KUKA KRL program: MyProgram_022().src

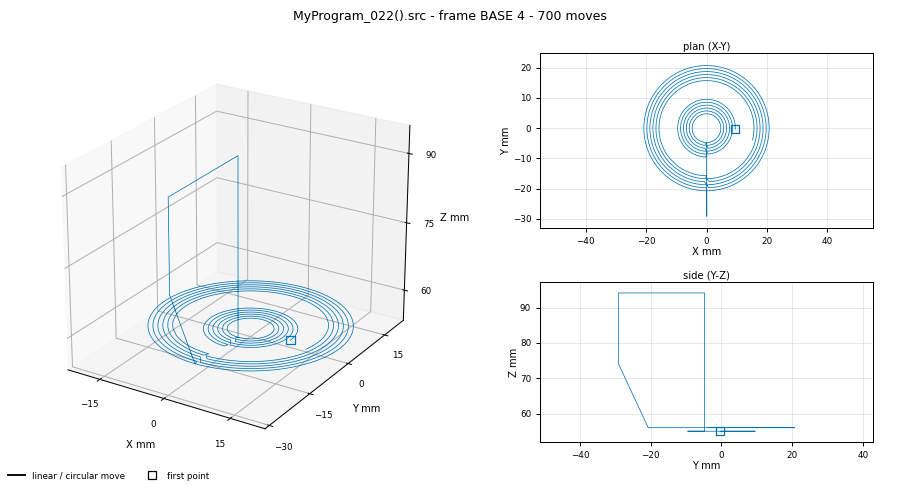
[picture p0: tool path of MyProgram_022().src in frame BASE 4, 700 of 700 moves have a stored position in this frame; points joined in program order, loops and branches not executed]
&ACCESS RVP
&REL 1
&PARAM TEMPLATE = C:\KRC\Roboter\Template\vorgabe
&PARAM EDITMASK = *
DEF MyProgram_022()
; ---- Setting reference (Base) ----
$BASE = BASE_DATA[4]

; --------------------------
; ---- Setting tool (TCP) ----
$TOOL = TOOL_DATA[3]
; --------------------------

$VEL.CP = VEL_APROX_PRINT
Startdeposition()
$VEL.CP = VEL_PRINT
LIN {X 9.5437,Y -0.3407,Z 55,A -8.3961,B 24.5035,C -3.2675,E1 24.8669,E2 -269.4642} C_DIS
LIN {X 9.52,Y 0.7548,Z 55,A -1.6453,B 24.5009,C -3.2888,E1 24.8659,E2 -276.2255} C_DIS
LIN {X 9.3724,Y 1.8321,Z 55,A 5.8885,B 24.4976,C -3.3147,E1 24.8622,E2 -283.7766} C_DIS
LIN {X 8.9196,Y 3.4119,Z 55,A 15.084,B 24.4945,C -3.3389,E1 24.8541,E2 -292.9776} C_DIS
LIN {X 8.1843,Y 4.9212,Z 55,A 24.5802,B 24.4915,C -3.3621,E1 24.8417,E2 -302.4789} C_DIS
LIN {X 7.5338,Y 5.8685,Z 55,A 31.3136,B 24.4895,C -3.3777,E1 24.8306,E2 -309.2166} C_DIS
LIN {X 6.8523,Y 6.6485,Z 55,A 37.0507,B 24.4881,C -3.3886,E1 24.8199,E2 -314.9542} C_DIS
LIN {X 6.0078,Y 7.4234,Z 55,A 44.3227,B 24.4861,C -3.4035,E1 24.8046,E2 -322.233} C_DIS
LIN {X 5.0818,Y 8.0855,Z 55,A 51.1975,B 24.4847,C -3.4144,E1 24.7887,E2 -329.1106} C_DIS
LIN {X 4.1712,Y 8.5908,Z 55,A 57.4744,B 24.4837,C -3.4223,E1 24.7731,E2 -335.3889} C_DIS
LIN {X 3.3474,Y 8.9438,Z 55,A 62.8052,B 24.483,C -3.4273,E1 24.7593,E2 -340.7196} C_DIS
LIN {X 2.409,Y 9.2406,Z 55,A 69.1697,B 24.4823,C -3.4329,E1 24.7422,E2 -347.0869} C_DIS
LIN {X 1.1691,Y 9.477,Z 55,A 76.1197,B 24.4823,C -3.4331,E1 24.723,E2 -354.0304} C_DIS
LIN {X 0.1545,Y 9.5485,Z 55,A 82.3576,B 24.4823,C -3.4331,E1 24.7056,E2 -360.2665} C_DIS
LIN {X -1.2836,Y 9.4632,Z 55,A 91.4292,B 24.4826,C -3.4303,E1 24.6804,E2 -369.3357} C_DIS
LIN {X -2.5093,Y 9.2143,Z 55,A 98.8876,B 24.4835,C -3.4234,E1 24.6602,E2 -376.7878} C_DIS
LIN {X -3.3779,Y 8.9324,Z 55,A 105.3226,B 24.4842,C -3.4184,E1 24.6434,E2 -383.2239} C_DIS
LIN {X -4.9252,Y 8.1819,Z 55,A 114.2089,B 24.4867,C -3.3995,E1 24.6215,E2 -392.0897} C_DIS
LIN {X -5.8293,Y 7.5644,Z 55,A 121.6467,B 24.4882,C -3.3875,E1 24.6048,E2 -399.525} C_DIS
LIN {X -6.7767,Y 6.7285,Z 55,A 128.6516,B 24.4905,C -3.3699,E1 24.5905,E2 -406.5164} C_DIS
LIN {X -7.5818,Y 5.8012,Z 55,A 134.4735,B 24.493,C -3.3508,E1 24.5801,E2 -412.319} C_DIS
LIN {X -8.0674,Y 5.1105,Z 55,A 141.4999,B 24.4946,C -3.338,E1 24.5691,E2 -419.3498} C_DIS
LIN {X -8.6788,Y 3.9781,Z 55,A 147.4247,B 24.4974,C -3.3158,E1 24.5615,E2 -425.2526} C_DIS
LIN {X -9.0093,Y 3.1669,Z 55,A 154.8449,B 24.4994,C -3.3005,E1 24.5541,E2 -432.6779} C_DIS
LIN {X -9.3639,Y 1.875,Z 55,A 161.7964,B 24.5025,C -3.2759,E1 24.5495,E2 -439.6111} C_DIS
LIN {X -9.529,Y 0.6276,Z 55,A 171.0146,B 24.5054,C -3.2526,E1 24.5469,E2 -448.8287} C_DIS
LIN {X -9.5121,Y -0.8487,Z 55,A 178.9892,B 24.5088,C -3.2253,E1 24.548,E2 -456.7858} C_DIS
LIN {X -9.3498,Y -1.944,Z 55,A -174.6947,B 24.5112,C -3.2053,E1 24.551,E2 -463.0913} C_DIS
LIN {X -9.078,Y -2.965,Z 55,A -167.6269,B 24.5135,C -3.187,E1 24.5566,E2 -470.1561} C_DIS
LIN {X -8.6807,Y -3.9802,Z 55,A -161.2388,B 24.5157,C -3.169,E1 24.5636,E2 -476.5362} C_DIS
LIN {X -8.1263,Y -5.0163,Z 55,A -154.1121,B 24.5179,C -3.1509,E1 24.5735,E2 -483.6566} C_DIS
LIN {X -7.4885,Y -5.9263,Z 55,A -147.3718,B 24.5198,C -3.1353,E1 24.5848,E2 -490.392} C_DIS
LIN {X -6.6668,Y -6.8377,Z 55,A -139.7416,B 24.5215,C -3.1203,E1 24.5996,E2 -498.0193} C_DIS
LIN {X -5.7118,Y -7.6497,Z 55,A -133.1323,B 24.5233,C -3.1057,E1 24.6139,E2 -504.6186} C_DIS
LIN {X -4.7809,Y -8.267,Z 55,A -125.9127,B 24.5243,C -3.0968,E1 24.631,E2 -511.8397} C_DIS
LIN {X -3.8134,Y -8.7552,Z 55,A -118.9983,B 24.5251,C -3.0904,E1 24.6485,E2 -518.7563} C_DIS
LIN {X -2.6205,Y -9.1833,Z 55,A -111.5476,B 24.5258,C -3.0845,E1 24.6683,E2 -526.2062} C_DIS
LIN {X -1.4624,Y -9.4371,Z 55,A -104.4401,B 24.5261,C -3.082,E1 24.6878,E2 -533.3153} C_DIS
LIN {X -0.2812,Y -9.5456,Z 55,A -97.8601,B 24.5263,C -3.0804,E1 24.7061,E2 -539.8939} C_DIS
LIN {X -0.2812,Y -9.5456,Z 55,A -97.8601,B 24.5263,C -3.0804,E1 24.7061,E2 -539.8939} C_DIS
Enddeposition()
LIN {X 0.0484,Y -8.5882,Z 55,A -96.4156,B 19.666,C -2.0295,E1 19.7657,E2 -540.06} C_DIS
Startdeposition()
$VEL.CP = VEL_PRINT
LIN {X -1.0617,Y -8.5255,Z 55,A -105.0334,B 19.6663,C -2.0274,E1 19.7417,E2 -531.431} C_DIS
LIN {X -2.1331,Y -8.3222,Z 55,A -111.7699,B 19.6658,C -2.0316,E1 19.7233,E2 -524.6964} C_DIS
LIN {X -2.9014,Y -8.0865,Z 55,A -117.4774,B 19.6655,C -2.0353,E1 19.7082,E2 -518.986} C_DIS
LIN {X -3.626,Y -7.7883,Z 55,A -122.789,B 19.6649,C -2.0407,E1 19.6947,E2 -513.6739} C_DIS
LIN {X -4.5351,Y -7.2969,Z 55,A -130.0587,B 19.664,C -2.0498,E1 19.6772,E2 -506.4028} C_DIS
LIN {X -5.617,Y -6.5006,Z 55,A -138.2989,B 19.6625,C -2.0653,E1 19.6591,E2 -498.1697} C_DIS
LIN {X -6.3065,Y -5.8281,Z 55,A -144.638,B 19.6612,C -2.0782,E1 19.6467,E2 -491.8342} C_DIS
LIN {X -6.8045,Y -5.2401,Z 55,A -149.8115,B 19.66,C -2.0896,E1 19.6376,E2 -486.6633} C_DIS
LIN {X -7.4508,Y -4.2776,Z 55,A -158.3349,B 19.658,C -2.1086,E1 19.6249,E2 -478.1405} C_DIS
LIN {X -7.8893,Y -3.4012,Z 55,A -165.4977,B 19.6562,C -2.1262,E1 19.6167,E2 -470.9797} C_DIS
LIN {X -8.3397,Y -2.0642,Z 55,A -174.2614,B 19.6535,C -2.1523,E1 19.6097,E2 -462.2282} C_DIS
LIN {X -8.5403,Y -0.9049,Z 55,A 179.7232,B 19.6512,C -2.1738,E1 19.6071,E2 -456.2308} C_DIS
LIN {X -8.5918,Y -0.0576,Z 55,A 171.3138,B 19.6492,C -2.1929,E1 19.6063,E2 -447.813} C_DIS
LIN {X -8.5069,Y 1.2012,Z 55,A 164.3732,B 19.6466,C -2.2167,E1 19.6081,E2 -440.8896} C_DIS
LIN {X -8.3384,Y 2.0688,Z 55,A 156.7921,B 19.6446,C -2.2355,E1 19.6128,E2 -433.307} C_DIS
LIN {X -7.8607,Y 3.4667,Z 55,A 148.6266,B 19.6416,C -2.2623,E1 19.6208,E2 -425.162} C_DIS
LIN {X -7.4985,Y 4.1927,Z 55,A 141.6224,B 19.6399,C -2.2779,E1 19.63,E2 -418.1563} C_DIS
LIN {X -6.649,Y 5.4408,Z 55,A 133.1113,B 19.6371,C -2.3025,E1 19.6439,E2 -409.665} C_DIS
LIN {X -6.1281,Y 6.021,Z 55,A 125.7768,B 19.6358,C -2.3146,E1 19.6581,E2 -402.3256} C_DIS
LIN {X -4.7675,Y 7.1472,Z 55,A 114.9917,B 19.6332,C -2.3374,E1 19.6819,E2 -391.5581} C_DIS
LIN {X -4.0838,Y 7.5577,Z 55,A 109.5222,B 19.6322,C -2.3457,E1 19.6953,E2 -386.0929} C_DIS
LIN {X -2.9018,Y 8.0863,Z 55,A 100.8347,B 19.631,C -2.3565,E1 19.7177,E2 -377.4126} C_DIS
LIN {X -1.6334,Y 8.434,Z 55,A 92.4272,B 19.6301,C -2.3643,E1 19.7405,E2 -369.0136} C_DIS
LIN {X -0.6223,Y 8.5687,Z 55,A 85.3058,B 19.6298,C -2.3669,E1 19.7602,E2 -361.8945} C_DIS
LIN {X 0.509,Y 8.5714,Z 55,A 78.3367,B 19.6296,C -2.3687,E1 19.7797,E2 -354.9324} C_DIS
LIN {X 1.2791,Y 8.4924,Z 55,A 73.1686,B 19.6297,C -2.3675,E1 19.794,E2 -349.7659} C_DIS
LIN {X 2.0387,Y 8.3424,Z 55,A 68.0068,B 19.63,C -2.3649,E1 19.808,E2 -344.6055} C_DIS
LIN {X 3.1694,Y 7.9849,Z 55,A 60.3912,B 19.6307,C -2.3592,E1 19.8281,E2 -336.9923} C_DIS
LIN {X 4.1301,Y 7.5333,Z 55,A 51.4713,B 19.6324,C -2.3444,E1 19.8503,E2 -328.0604} C_DIS
LIN {X 5.3942,Y 6.6869,Z 55,A 44.1822,B 19.633,C -2.3388,E1 19.8669,E2 -320.7874} C_DIS
LIN {X 6.1554,Y 5.9934,Z 55,A 35.7616,B 19.6352,C -2.3192,E1 19.8841,E2 -312.3536} C_DIS
LIN {X 6.7864,Y 5.2679,Z 55,A 28.6991,B 19.6372,C -2.3022,E1 19.8965,E2 -305.2831} C_DIS
LIN {X 7.5014,Y 4.1881,Z 55,A 21.2861,B 19.6389,C -2.2866,E1 19.9074,E2 -297.8727} C_DIS
LIN {X 7.8951,Y 3.3879,Z 55,A 15.4697,B 19.6406,C -2.2715,E1 19.9143,E2 -292.0525} C_DIS
LIN {X 8.2732,Y 2.3161,Z 55,A 7.2455,B 19.6433,C -2.2472,E1 19.9215,E2 -283.8168} C_DIS
LIN {X 8.491,Y 1.2828,Z 55,A 0.8671,B 19.6452,C -2.2301,E1 19.9248,E2 -277.4363} C_DIS
LIN {X 8.5896,Y 0.1713,Z 55,A -7.1351,B 19.6479,C -2.2051,E1 19.9261,E2 -269.4218} C_DIS
LIN {X 8.5419,Y -0.9196,Z 55,A -14.0427,B 19.65,C -2.1853,E1 19.9248,E2 -262.5087} C_DIS
LIN {X 8.3771,Y -1.906,Z 55,A -21.1303,B 19.6523,C -2.1634,E1 19.9209,E2 -255.4101} C_DIS
LIN {X 8.0567,Y -2.9832,Z 55,A -28.7401,B 19.6547,C -2.1411,E1 19.9142,E2 -247.7903} C_DIS
LIN {X 7.587,Y -4.0309,Z 55,A -35.9207,B 19.6566,C -2.1223,E1 19.9054,E2 -240.6039} C_DIS
LIN {X 6.9736,Y -5.0179,Z 55,A -45.1996,B 19.6594,C -2.0953,E1 19.8908,E2 -231.3045} C_DIS
LIN {X 5.6333,Y -6.4865,Z 55,A -56.5929,B 19.6616,C -2.0736,E1 19.8684,E2 -219.91} C_DIS
LIN {X 4.5247,Y -7.3028,Z 55,A -67.0354,B 19.6638,C -2.0518,E1 19.8443,E2 -209.4489} C_DIS
LIN {X 3.1306,Y -8.0001,Z 55,A -77.5224,B 19.6653,C -2.0372,E1 19.8175,E2 -198.952} C_DIS
LIN {X 1.7735,Y -8.4063,Z 55,A -86.5252,B 19.666,C -2.03,E1 19.7932,E2 -189.9452} C_DIS
LIN {X 0.493,Y -8.5769,Z 55,A -94.5546,B 19.6662,C -2.0275,E1 19.7709,E2 -181.9148} C_DIS
LIN {X 0.493,Y -8.5769,Z 55,A -94.5546,B 19.6662,C -2.0275,E1 19.7709,E2 -181.9148} C_DIS
Enddeposition()
LIN {X -0.0072,Y -7.6328,Z 55,A -91.0932,B 14.7927,C -1.2124,E1 14.8521,E2 -184.2665} C_DIS
Startdeposition()
$VEL.CP = VEL_PRINT
LIN {X 1.7414,Y -7.4315,Z 55,A -79.0266,B 14.7923,C -1.2183,E1 14.8852,E2 -196.3334} C_DIS
LIN {X 3.0947,Y -6.9771,Z 55,A -69.7981,B 14.7916,C -1.2267,E1 14.9093,E2 -205.56} C_DIS
LIN {X 3.8118,Y -6.6129,Z 55,A -64.1101,B 14.7909,C -1.2346,E1 14.9234,E2 -211.2506} C_DIS
LIN {X 4.7649,Y -5.9629,Z 55,A -52.7906,B 14.7889,C -1.2595,E1 14.9488,E2 -222.596} C_DIS
LIN {X 5.9068,Y -4.8341,Z 55,A -40.8403,B 14.7866,C -1.2863,E1 14.9711,E2 -234.5569} C_DIS
LIN {X 6.931,Y -3.1967,Z 55,A -28.3133,B 14.7841,C -1.3158,E1 14.9882,E2 -247.0842} C_DIS
LIN {X 7.2359,Y -2.4292,Z 55,A -21.4776,B 14.7823,C -1.3357,E1 14.9947,E2 -253.9303} C_DIS
LIN {X 7.5213,Y -1.3,Z 55,A -13.0631,B 14.7802,C -1.3594,E1 14.9996,E2 -262.3507} C_DIS
LIN {X 7.6295,Y -0.2251,Z 55,A -5.4007,B 14.7783,C -1.381,E1 15.001,E2 -270.0173} C_DIS
LIN {X 7.5606,Y 1.0475,Z 55,A 4.7584,B 14.7755,C -1.4111,E1 14.9984,E2 -280.188} C_DIS
LIN {X 7.3346,Y 2.1124,Z 55,A 12.6105,B 14.7735,C -1.4325,E1 14.993,E2 -288.0437} C_DIS
LIN {X 6.904,Y 3.2548,Z 55,A 21.287,B 14.7714,C -1.4546,E1 14.9837,E2 -296.7226} C_DIS
LIN {X 6.4679,Y 4.053,Z 55,A 28.2666,B 14.7697,C -1.4719,E1 14.9738,E2 -303.7065} C_DIS
LIN {X 5.86,Y 4.8857,Z 55,A 35.0672,B 14.7683,C -1.4858,E1 14.9623,E2 -310.5044} C_DIS
LIN {X 5.403,Y 5.3885,Z 55,A 40.3436,B 14.7672,C -1.4968,E1 14.9521,E2 -315.7833} C_DIS
LIN {X 4.5877,Y 6.1003,Z 55,A 48.6669,B 14.7657,C -1.5118,E1 14.9342,E2 -324.1091} C_DIS
LIN {X 3.6389,Y 6.7096,Z 55,A 58.0991,B 14.7643,C -1.5264,E1 14.9116,E2 -333.5471} C_DIS
LIN {X 2.5598,Y 7.1908,Z 55,A 66.5015,B 14.7635,C -1.534,E1 14.8898,E2 -341.9457} C_DIS
LIN {X 1.3106,Y 7.5193,Z 55,A 76.1296,B 14.763,C -1.5391,E1 14.8636,E2 -351.5707} C_DIS
LIN {X 0.2159,Y 7.6256,Z 55,A 83.5677,B 14.763,C -1.5388,E1 14.8429,E2 -359.0012} C_DIS
LIN {X -0.8816,Y 7.5817,Z 55,A 91.5987,B 14.7633,C -1.5362,E1 14.8206,E2 -367.0266} C_DIS
LIN {X -1.6402,Y 7.4545,Z 55,A 98.3351,B 14.7636,C -1.5333,E1 14.8021,E2 -373.7643} C_DIS
LIN {X -2.5722,Y 7.1863,Z 55,A 105.734,B 14.7643,C -1.5262,E1 14.7825,E2 -381.1586} C_DIS
LIN {X -3.6086,Y 6.7255,Z 55,A 113.7963,B 14.7654,C -1.5147,E1 14.7623,E2 -389.2118} C_DIS
LIN {X -4.467,Y 6.1826,Z 55,A 121.4415,B 14.7667,C -1.5019,E1 14.7445,E2 -396.8508} C_DIS
LIN {X -5.1004,Y 5.6736,Z 55,A 127.6071,B 14.7679,C -1.49,E1 14.7314,E2 -403.0111} C_DIS
LIN {X -5.6752,Y 5.0991,Z 55,A 133.8696,B 14.7692,C -1.4766,E1 14.7194,E2 -409.2685} C_DIS
LIN {X -6.305,Y 4.302,Z 55,A 141.9263,B 14.771,C -1.4579,E1 14.7061,E2 -417.3199} C_DIS
LIN {X -6.8966,Y 3.2703,Z 55,A 151.3038,B 14.7733,C -1.434,E1 14.6939,E2 -426.6908} C_DIS
LIN {X -7.3324,Y 2.1063,Z 55,A 159.9509,B 14.7757,C -1.409,E1 14.6862,E2 -435.3257} C_DIS
LIN {X -7.5725,Y 0.9578,Z 55,A 168.9473,B 14.7781,C -1.3833,E1 14.6818,E2 -444.3148} C_DIS
LIN {X -7.6314,Y 0.1435,Z 55,A 175.5205,B 14.7797,C -1.3649,E1 14.681,E2 -450.8849} C_DIS
LIN {X -7.5817,Y -0.8637,Z 55,A -177.4519,B 14.7816,C -1.3438,E1 14.6825,E2 -457.9037} C_DIS
LIN {X -7.4779,Y -1.5155,Z 55,A -172.4272,B 14.7829,C -1.3297,E1 14.685,E2 -462.9251} C_DIS
LIN {X -7.3187,Y -2.1561,Z 55,A -167.5507,B 14.7841,C -1.3161,E1 14.6886,E2 -467.7976} C_DIS
LIN {X -7.1055,Y -2.7807,Z 55,A -162.5731,B 14.7852,C -1.3027,E1 14.6933,E2 -472.7722} C_DIS
LIN {X -6.6528,Y -3.7418,Z 55,A -153.6372,B 14.787,C -1.2816,E1 14.7047,E2 -481.7088} C_DIS
LIN {X -6.2826,Y -4.3348,Z 55,A -147.702,B 14.7881,C -1.2688,E1 14.714,E2 -487.6455} C_DIS
LIN {X -5.4108,Y -5.3837,Z 55,A -138.4398,B 14.7898,C -1.2482,E1 14.7312,E2 -496.899} C_DIS
LIN {X -4.5966,Y -6.0937,Z 55,A -129.9493,B 14.791,C -1.2341,E1 14.7496,E2 -505.3903} C_DIS
LIN {X -3.8307,Y -6.602,Z 55,A -122.8606,B 14.7918,C -1.2244,E1 14.7664,E2 -512.4797} C_DIS
LIN {X -2.8961,Y -7.0619,Z 55,A -115.5853,B 14.7924,C -1.2159,E1 14.7849,E2 -519.7524} C_DIS
LIN {X -2.0683,Y -7.3434,Z 55,A -109.3433,B 14.7929,C -1.2108,E1 14.8015,E2 -525.9939} C_DIS
LIN {X -1.0315,Y -7.5626,Z 55,A -99.7498,B 14.7929,C -1.2099,E1 14.8279,E2 -535.6} C_DIS
LIN {X -0.0072,Y -7.6328,Z 55,A -95.8758,B 14.7934,C -1.2042,E1 14.8386,E2 -539.4534} C_DIS
Enddeposition()
LIN {X -0.0072,Y -7.6328,Z 55,A -95.8758,B 14.7934,C -1.2042,E1 14.8386,E2 -539.4534} C_DIS
Startdeposition()
$VEL.CP = VEL_PRINT
LIN {X -0.5513,Y -6.6453,Z 55,A -99.3031,B 9.8862,C -0.5743,E1 9.8872,E2 -534.9699} C_DIS
LIN {X -1.4265,Y -6.52,Z 55,A -108.8863,B 9.8861,C -0.5765,E1 9.8609,E2 -525.3735} C_DIS
LIN {X -2.7177,Y -6.0958,Z 55,A -119.3612,B 9.8855,C -0.5868,E1 9.8336,E2 -514.9021} C_DIS
LIN {X -3.4112,Y -5.7368,Z 55,A -126.4444,B 9.885,C -0.5957,E1 9.8164,E2 -507.8162} C_DIS
LIN {X -4.2862,Y -5.1161,Z 55,A -135.5205,B 9.884,C -0.6107,E1 9.7963,E2 -498.7408} C_DIS
LIN {X -5.0009,Y -4.4131,Z 55,A -143.9478,B 9.883,C -0.6275,E1 9.78,E2 -490.3155} C_DIS
LIN {X -5.6735,Y -3.5155,Z 55,A -154.2169,B 9.8815,C -0.6504,E1 9.7637,E2 -480.0455} C_DIS
LIN {X -6.1829,Y -2.5134,Z 55,A -164.5095,B 9.8798,C -0.6761,E1 9.7518,E2 -469.7535} C_DIS
LIN {X -6.5159,Y -1.4238,Z 55,A -173.0169,B 9.8782,C -0.7003,E1 9.7455,E2 -461.2563} C_DIS
LIN {X -6.629,Y -0.7484,Z 55,A -179.2232,B 9.8769,C -0.7174,E1 9.7431,E2 -455.0517} C_DIS
LIN {X -6.6704,Y -0.0648,Z 55,A 174.6774,B 9.8757,C -0.7346,E1 9.7425,E2 -448.9549} C_DIS
LIN {X -6.6273,Y 0.7901,Z 55,A 166.5401,B 9.874,C -0.757,E1 9.7445,E2 -440.8189} C_DIS
LIN {X -6.3943,Y 1.901,Z 55,A 156.9959,B 9.872,C -0.7837,E1 9.7508,E2 -431.2824} C_DIS
LIN {X -6.1141,Y 2.6653,Z 55,A 150.0872,B 9.8705,C -0.8022,E1 9.758,E2 -424.3791} C_DIS
LIN {X -5.7439,Y 3.3901,Z 55,A 142.9913,B 9.869,C -0.82,E1 9.7675,E2 -417.288} C_DIS
LIN {X -5.2892,Y 4.0652,Z 55,A 135.855,B 9.8677,C -0.8365,E1 9.7791,E2 -410.1563} C_DIS
LIN {X -4.7541,Y 4.6787,Z 55,A 128.7619,B 9.8664,C -0.8515,E1 9.7925,E2 -403.0681} C_DIS
LIN {X -3.8851,Y 5.427,Z 55,A 117.8688,B 9.8648,C -0.8702,E1 9.8164,E2 -392.178} C_DIS
LIN {X -2.9088,Y 6.0071,Z 55,A 108.4824,B 9.8636,C -0.8834,E1 9.8394,E2 -382.7998} C_DIS
LIN {X -1.9263,Y 6.3903,Z 55,A 99.5045,B 9.8628,C -0.8922,E1 9.863,E2 -373.828} C_DIS
LIN {X -0.8857,Y 6.6117,Z 55,A 92.459,B 9.8623,C -0.898,E1 9.8823,E2 -366.7966} C_DIS
LIN {X 0.1331,Y 6.6728,Z 55,A 80.869,B 9.8623,C -0.8972,E1 9.9146,E2 -355.1986} C_DIS
LIN {X 1.2683,Y 6.5482,Z 55,A 72.5953,B 9.8625,C -0.8955,E1 9.9374,E2 -346.9354} C_DIS
LIN {X 1.9117,Y 6.3913,Z 55,A 66.8902,B 9.8629,C -0.8915,E1 9.9528,E2 -341.2319} C_DIS
LIN {X 3.0336,Y 5.945,Z 55,A 55.2257,B 9.8641,C -0.8775,E1 9.9826,E2 -329.5632} C_DIS
LIN {X 3.8966,Y 5.4188,Z 55,A 46.0037,B 9.8654,C -0.8626,E1 10.0038,E2 -320.3392} C_DIS
LIN {X 4.9697,Y 4.4553,Z 55,A 34.8499,B 9.8672,C -0.8418,E1 10.026,E2 -309.1902} C_DIS
LIN {X 5.472,Y 3.8144,Z 55,A 28.6234,B 9.8683,C -0.8284,E1 10.0363,E2 -302.9662} C_DIS
LIN {X 5.818,Y 3.2625,Z 55,A 23.1367,B 9.8694,C -0.8152,E1 10.0442,E2 -297.4784} C_DIS
LIN {X 6.1096,Y 2.68,Z 55,A 17.5975,B 9.8706,C -0.8012,E1 10.0507,E2 -291.9376} C_DIS
LIN {X 6.3418,Y 2.0713,Z 55,A 12.2288,B 9.8717,C -0.7871,E1 10.0557,E2 -286.5677} C_DIS
LIN {X 6.582,Y 1.1054,Z 55,A 3.0945,B 9.8737,C -0.7613,E1 10.0611,E2 -277.4261} C_DIS
LIN {X 6.6738,Y 0.0305,Z 55,A -7.2201,B 9.8759,C -0.7312,E1 10.0623,E2 -267.1005} C_DIS
LIN {X 6.5795,Y -1.1203,Z 55,A -18.0928,B 9.8782,C -0.6997,E1 10.0578,E2 -256.2161} C_DIS
LIN {X 6.045,Y -2.829,Z 55,A -31.9199,B 9.8807,C -0.6638,E1 10.044,E2 -242.3863} C_DIS
LIN {X 5.2656,Y -4.1012,Z 55,A -43.2424,B 9.8824,C -0.6376,E1 10.0264,E2 -231.0624} C_DIS
LIN {X 4.795,Y -4.6426,Z 55,A -51.3115,B 9.8835,C -0.6188,E1 10.0109,E2 -222.9781} C_DIS
LIN {X 3.4915,Y -5.6883,Z 55,A -63.9968,B 9.8848,C -0.5978,E1 9.9822,E2 -210.2916} C_DIS
LIN {X 2.6709,Y -6.1105,Z 55,A -71.3878,B 9.8854,C -0.5883,E1 9.9637,E2 -202.8983} C_DIS
LIN {X 1.9793,Y -6.3683,Z 55,A -77.5808,B 9.8858,C -0.582,E1 9.9473,E2 -196.7021} C_DIS
LIN {X 1.2637,Y -6.5499,Z 55,A -84.0144,B 9.886,C -0.5772,E1 9.9298,E2 -190.2642} C_DIS
LIN {X 0.5322,Y -6.6495,Z 55,A -90.4765,B 9.8862,C -0.5743,E1 9.9118,E2 -183.7981} C_DIS
LIN {X 0.5322,Y -6.6495,Z 55,A -90.4765,B 9.8862,C -0.5743,E1 9.9118,E2 -183.7981} C_DIS
Enddeposition()
LIN {X -0.0091,Y -5.7118,Z 55,A -2.8836,B 0,C 0,E1 0.1598,E2 -269.9283} C_DIS
Startdeposition()
$VEL.CP = VEL_PRINT
LIN {X 0.9619,Y -5.6271,Z 55,A -2.8445,B 0,C 0,E1 0.1598,E2 -269.9283} C_DIS
LIN {X 1.7206,Y -5.4461,Z 55,A -2.8089,B 0,C 0,E1 0.1598,E2 -269.9282} C_DIS
LIN {X 2.4463,Y -5.1598,Z 55,A -2.77,B 0,C 0,E1 0.1598,E2 -269.9282} C_DIS
LIN {X 3.127,Y -4.7788,Z 55,A -2.7288,B 0,C 0,E1 0.1598,E2 -269.9282} C_DIS
LIN {X 4.0215,Y -4.0615,Z 55,A -2.6651,B 0,C 0,E1 0.1598,E2 -269.9282} C_DIS
LIN {X 4.6904,Y -3.2657,Z 55,A -2.6064,B 0,C 0,E1 0.1598,E2 -269.9282} C_DIS
LIN {X 5.1397,Y -2.4895,Z 55,A -2.5568,B 0,C 0,E1 0.1598,E2 -269.9282} C_DIS
LIN {X 5.4534,Y -1.6925,Z 55,A -2.5112,B 0,C 0,E1 0.1598,E2 -269.9282} C_DIS
LIN {X 5.6446,Y -0.8577,Z 55,A -2.4685,B 0,C 0,E1 0.1598,E2 -269.9282} C_DIS
LIN {X 5.7096,Y -0.0038,Z 55,A -2.4296,B 0,C 0,E1 0.1598,E2 -269.9281} C_DIS
LIN {X 5.6161,Y 1.0625,Z 55,A -2.3872,B 0,C 0,E1 0.1598,E2 -269.9284} C_DIS
LIN {X 5.3029,Y 2.1179,Z 55,A -2.3537,B 0,C 0,E1 0.1598,E2 -269.9283} C_DIS
LIN {X 4.959,Y 2.8274,Z 55,A -2.3364,B 0,C 0,E1 0.1598,E2 -269.9279} C_DIS
LIN {X 4.5235,Y 3.4846,Z 55,A -2.3245,B 0,C 0,E1 0.1598,E2 -269.9278} C_DIS
LIN {X 4.0015,Y 4.0757,Z 55,A -2.3186,B 0,C 0,E1 0.1598,E2 -269.9278} C_DIS
LIN {X 3.4014,Y 4.5875,Z 55,A -2.3189,B 0,C 0,E1 0.1598,E2 -269.9277} C_DIS
LIN {X 2.7366,Y 5.0113,Z 55,A -2.3254,B 0,C 0,E1 0.1598,E2 -269.9277} C_DIS
LIN {X 1.7186,Y 5.4511,Z 55,A -2.3442,B 0,C 0,E1 0.1598,E2 -269.9277} C_DIS
LIN {X 0.5579,Y 5.6885,Z 55,A -2.377,B 0,C 0,E1 0.1598,E2 -269.9277} C_DIS
LIN {X -0.385,Y 5.6987,Z 55,A -2.4114,B 0,C 0,E1 0.1598,E2 -269.9277} C_DIS
LIN {X -1.1326,Y 5.5975,Z 55,A -2.4432,B 0,C 0,E1 0.1598,E2 -269.9277} C_DIS
LIN {X -1.8604,Y 5.4,Z 55,A -2.4785,B 0,C 0,E1 0.1598,E2 -269.9277} C_DIS
LIN {X -2.5543,Y 5.1047,Z 55,A -2.5166,B 0,C 0,E1 0.1598,E2 -269.9278} C_DIS
LIN {X -3.2057,Y 4.7249,Z 55,A -2.5567,B 0,C 0,E1 0.1598,E2 -269.9279} C_DIS
LIN {X -3.8016,Y 4.2624,Z 55,A -2.5982,B 0,C 0,E1 0.1598,E2 -269.928} C_DIS
LIN {X -4.3298,Y 3.7239,Z 55,A -2.6405,B 0,C 0,E1 0.1598,E2 -269.928} C_DIS
LIN {X -4.7804,Y 3.1193,Z 55,A -2.6827,B 0,C 0,E1 0.1598,E2 -269.9282} C_DIS
LIN {X -5.1513,Y 2.4628,Z 55,A -2.7242,B 0,C 0,E1 0.1598,E2 -269.9282} C_DIS
LIN {X -5.431,Y 1.7624,Z 55,A -2.7641,B 0,C 0,E1 0.1598,E2 -269.9284} C_DIS
LIN {X -5.6177,Y 1.0317,Z 55,A -2.802,B 0,C 0,E1 0.1598,E2 -269.9284} C_DIS
LIN {X -5.7035,Y 0.2823,Z 55,A -2.8369,B 0,C 0,E1 0.1598,E2 -269.9285} C_DIS
LIN {X -5.69,Y -0.4718,Z 55,A -2.8684,B 0,C 0,E1 0.1598,E2 -269.9285} C_DIS
LIN {X -5.541,Y -1.4026,Z 55,A -2.9022,B 0,C 0,E1 0.1598,E2 -269.9288} C_DIS
LIN {X -4.946,Y -2.8649,Z 55,A -2.9418,B 0,C 0,E1 0.1598,E2 -269.9295} C_DIS
LIN {X -4.4029,Y -3.645,Z 55,A -2.9555,B 0,C 0,E1 0.1598,E2 -269.9291} C_DIS
LIN {X -3.4666,Y -4.5443,Z 55,A -2.9596,B 0,C 0,E1 0.1598,E2 -269.9288} C_DIS
LIN {X -2.4461,Y -5.1659,Z 55,A -2.9488,B 0,C 0,E1 0.1598,E2 -269.9286} C_DIS
LIN {X -1.3162,Y -5.5622,Z 55,A -2.9243,B 0,C 0,E1 0.1598,E2 -269.9284} C_DIS
LIN {X -0.5027,Y -5.6894,Z 55,A -2.9,B 0,C 0,E1 0.1598,E2 -269.9284} C_DIS
LIN {X -0.5027,Y -5.6894,Z 55,A -2.9,B 0,C 0,E1 0.1598,E2 -269.9283} C_DIS
Enddeposition()
LIN {X -0.0164,Y -4.7573,Z 55,A -2.841,B 0,C 0,E1 0.1598,E2 -269.9295} C_DIS
Startdeposition()
$VEL.CP = VEL_PRINT
LIN {X -0.8506,Y -4.6765,Z 55,A -2.8694,B 0,C 0,E1 0.1598,E2 -269.9283} C_DIS
LIN {X -1.5,Y -4.5096,Z 55,A -2.8862,B 0,C 0,E1 0.1598,E2 -269.9283} C_DIS
LIN {X -2.1197,Y -4.2534,Z 55,A -2.898,B 0,C 0,E1 0.1598,E2 -269.9283} C_DIS
LIN {X -2.6968,Y -3.9121,Z 55,A -2.9046,B 0,C 0,E1 0.1598,E2 -269.9283} C_DIS
LIN {X -3.2199,Y -3.4929,Z 55,A -2.906,B 0,C 0,E1 0.1598,E2 -269.9284} C_DIS
LIN {X -3.6802,Y -3.0058,Z 55,A -2.9021,B 0,C 0,E1 0.1598,E2 -269.9284} C_DIS
LIN {X -4.0666,Y -2.458,Z 55,A -2.893,B 0,C 0,E1 0.1598,E2 -269.9284} C_DIS
LIN {X -4.372,Y -1.8613,Z 55,A -2.8788,B 0,C 0,E1 0.1598,E2 -269.9284} C_DIS
LIN {X -4.5913,Y -1.2278,Z 55,A -2.86,B 0,C 0,E1 0.1598,E2 -269.9284} C_DIS
LIN {X -4.7168,Y -0.5691,Z 55,A -2.8366,B 0,C 0,E1 0.1598,E2 -269.9284} C_DIS
LIN {X -4.7518,Y 0.1003,Z 55,A -2.8094,B 0,C 0,E1 0.1598,E2 -269.9284} C_DIS
LIN {X -4.6905,Y 0.768,Z 55,A -2.7788,B 0,C 0,E1 0.1598,E2 -269.9284} C_DIS
LIN {X -4.5362,Y 1.4205,Z 55,A -2.7455,B 0,C 0,E1 0.1598,E2 -269.9284} C_DIS
LIN {X -4.2904,Y 2.0444,Z 55,A -2.71,B 0,C 0,E1 0.1598,E2 -269.9282} C_DIS
LIN {X -3.9574,Y 2.6262,Z 55,A -2.673,B 0,C 0,E1 0.1598,E2 -269.9282} C_DIS
LIN {X -3.5516,Y 3.1598,Z 55,A -2.6355,B 0,C 0,E1 0.1598,E2 -269.9281} C_DIS
LIN {X -3.0711,Y 3.6275,Z 55,A -2.5979,B 0,C 0,E1 0.1598,E2 -269.9281} C_DIS
LIN {X -2.5298,Y 4.0232,Z 55,A -2.5612,B 0,C 0,E1 0.1598,E2 -269.9279} C_DIS
LIN {X -1.9382,Y 4.3386,Z 55,A -2.526,B 0,C 0,E1 0.1598,E2 -269.9279} C_DIS
LIN {X -1.3083,Y 4.568,Z 55,A -2.4931,B 0,C 0,E1 0.1598,E2 -269.9278} C_DIS
LIN {X -0.6525,Y 4.7067,Z 55,A -2.4631,B 0,C 0,E1 0.1598,E2 -269.9278} C_DIS
LIN {X 0.0164,Y 4.7515,Z 55,A -2.4365,B 0,C 0,E1 0.1598,E2 -269.9277} C_DIS
LIN {X 0.6849,Y 4.7021,Z 55,A -2.414,B 0,C 0,E1 0.1598,E2 -269.9277} C_DIS
LIN {X 1.3398,Y 4.5588,Z 55,A -2.3959,B 0,C 0,E1 0.1598,E2 -269.9277} C_DIS
LIN {X 1.9677,Y 4.3241,Z 55,A -2.3827,B 0,C 0,E1 0.1598,E2 -269.9277} C_DIS
LIN {X 2.5574,Y 4.0054,Z 55,A -2.3745,B 0,C 0,E1 0.1598,E2 -269.9277} C_DIS
LIN {X 3.096,Y 3.6061,Z 55,A -2.3717,B 0,C 0,E1 0.1598,E2 -269.9277} C_DIS
LIN {X 3.5733,Y 3.1352,Z 55,A -2.3741,B 0,C 0,E1 0.1598,E2 -269.9277} C_DIS
LIN {X 3.9773,Y 2.5999,Z 55,A -2.382,B 0,C 0,E1 0.1598,E2 -269.9277} C_DIS
LIN {X 4.3039,Y 2.0145,Z 55,A -2.3949,B 0,C 0,E1 0.1598,E2 -269.9278} C_DIS
LIN {X 4.546,Y 1.3893,Z 55,A -2.4127,B 0,C 0,E1 0.1598,E2 -269.9278} C_DIS
LIN {X 4.6955,Y 0.7357,Z 55,A -2.435,B 0,C 0,E1 0.1598,E2 -269.9279} C_DIS
LIN {X 4.7525,Y 0.0675,Z 55,A -2.4615,B 0,C 0,E1 0.1598,E2 -269.9279} C_DIS
LIN {X 4.7136,Y -0.6018,Z 55,A -2.4915,B 0,C 0,E1 0.1598,E2 -269.928} C_DIS
LIN {X 4.5819,Y -1.2591,Z 55,A -2.5244,B 0,C 0,E1 0.1598,E2 -269.928} C_DIS
LIN {X 4.359,Y -1.8913,Z 55,A -2.5596,B 0,C 0,E1 0.1598,E2 -269.928} C_DIS
LIN {X 4.0496,Y -2.486,Z 55,A -2.5964,B 0,C 0,E1 0.1598,E2 -269.928} C_DIS
LIN {X 3.6587,Y -3.0304,Z 55,A -2.634,B 0,C 0,E1 0.1598,E2 -269.928} C_DIS
LIN {X 3.1965,Y -3.516,Z 55,A -2.6717,B 0,C 0,E1 0.1598,E2 -269.9281} C_DIS
LIN {X 2.6698,Y -3.9308,Z 55,A -2.7088,B 0,C 0,E1 0.1598,E2 -269.9281} C_DIS
LIN {X 2.0903,Y -4.268,Z 55,A -2.7445,B 0,C 0,E1 0.1598,E2 -269.9281} C_DIS
LIN {X 1.469,Y -4.5201,Z 55,A -2.7781,B 0,C 0,E1 0.1598,E2 -269.9281} C_DIS
LIN {X 0.8184,Y -4.6823,Z 55,A -2.8089,B 0,C 0,E1 0.1598,E2 -269.9281} C_DIS
LIN {X -0.0164,Y -4.7573,Z 55,A -2.8427,B 0,C 0,E1 0.1598,E2 -269.9282} C_DIS
Enddeposition()
LIN {X -0.0164,Y -4.7573,Z 60,A -2.8323,B 0,C 0,E1 0.1598,E2 -269.928} C_DIS
LIN {X -0.0164,Y -4.7571,Z 75,A -2.8055,B 0,C 0,E1 0.1598,E2 -269.927} C_DIS
LIN {X -0.0164,Y -4.7571,Z 94.1262,A -2.7793,B 0,C 0,E1 0.1598,E2 -269.9267} C_DIS
LIN {X 0.0643,Y -29.1728,Z 94.1262,A -97.2324,B 24.8219,C -3.0777,E1 25.0005,E2 -180.429} C_DIS
LIN {X 0.0643,Y -29.1728,Z 74.1262,A -96.9044,B 24.8376,C -2.94,E1 25.0005,E2 -180.429} C_DIS
LIN {X 0.0569,Y -22.8335,Z 60.5315,A -96.9447,B 24.8357,C -2.9569,E1 25.0005,E2 -180.429} C_DIS
LIN {X 0.0545,Y -20.7204,Z 56,A -96.9596,B 24.835,C -2.9632,E1 25.0005,E2 -180.429} C_DIS
Startdeposition()
$VEL.CP = VEL_PRINT
LIN {X 1.2873,Y -20.6848,Z 56,A -92.294,B 24.8338,C -2.9734,E1 25.0136,E2 -185.1177} C_DIS
LIN {X 3.0514,Y -20.4994,Z 56,A -87.4914,B 24.8336,C -2.9757,E1 25.0269,E2 -189.9219} C_DIS
LIN {X 4.6788,Y -20.1899,Z 56,A -82.799,B 24.833,C -2.9805,E1 25.0397,E2 -194.6198} C_DIS
LIN {X 6.3703,Y -19.7216,Z 56,A -77.9231,B 24.8324,C -2.9861,E1 25.0528,E2 -199.5004} C_DIS
LIN {X 7.9462,Y -19.1409,Z 56,A -73.5263,B 24.8319,C -2.9903,E1 25.0642,E2 -203.8974} C_DIS
LIN {X 9.4639,Y -18.4379,Z 56,A -68.7364,B 24.831,C -2.999,E1 25.0762,E2 -208.6953} C_DIS
LIN {X 11.0059,Y -17.5611,Z 56,A -63.8256,B 24.83,C -3.0078,E1 25.088,E2 -213.6119} C_DIS
LIN {X 12.456,Y -16.5641,Z 56,A -58.9873,B 24.8289,C -3.0173,E1 25.099,E2 -218.4557} C_DIS
LIN {X 13.8006,Y -15.4617,Z 56,A -54.1932,B 24.8277,C -3.0278,E1 25.1092,E2 -223.2559} C_DIS
LIN {X 15.0293,Y -14.2706,Z 56,A -49.5505,B 24.8265,C -3.0382,E1 25.1183,E2 -227.9035} C_DIS
LIN {X 16.1542,Y -12.9835,Z 56,A -44.8179,B 24.8251,C -3.0502,E1 25.1268,E2 -232.6429} C_DIS
LIN {X 17.2,Y -11.5623,Z 56,A -39.9191,B 24.8236,C -3.0634,E1 25.1347,E2 -237.5491} C_DIS
LIN {X 18.0989,Y -10.0971,Z 56,A -35.2338,B 24.8221,C -3.0761,E1 25.1413,E2 -242.2403} C_DIS
LIN {X 18.8655,Y -8.5803,Z 56,A -30.7037,B 24.8207,C -3.088,E1 25.1467,E2 -246.7744} C_DIS
LIN {X 19.4528,Y -7.1494,Z 56,A -26.3854,B 24.8192,C -3.1012,E1 25.1511,E2 -251.0999} C_DIS
LIN {X 19.9411,Y -5.6456,Z 56,A -21.9648,B 24.8176,C -3.115,E1 25.1547,E2 -255.528} C_DIS
LIN {X 20.3331,Y -4.0119,Z 56,A -17.4801,B 24.8161,C -3.1277,E1 25.1573,E2 -260.0168} C_DIS
LIN {X 20.5717,Y -2.5177,Z 56,A -13.1742,B 24.8144,C -3.142,E1 25.159,E2 -264.3311} C_DIS
LIN {X 20.7114,Y -0.7464,Z 56,A -8.943,B 24.8134,C -3.1505,E1 25.1597,E2 -268.5573} C_DIS
LIN {X 20.7189,Y 0.5147,Z 56,A -4.8529,B 24.8113,C -3.1674,E1 25.1597,E2 -272.6631} C_DIS
LIN {X 20.5986,Y 2.2843,Z 56,A -0.1749,B 24.8098,C -3.1802,E1 25.1585,E2 -277.3438} C_DIS
LIN {X 20.3685,Y 3.8281,Z 56,A 4.2815,B 24.8081,C -3.1947,E1 25.1564,E2 -281.8084} C_DIS
LIN {X 19.974,Y 5.5276,Z 56,A 9.0641,B 24.8064,C -3.2086,E1 25.1531,E2 -286.5964} C_DIS
LIN {X 19.4261,Y 7.2209,Z 56,A 13.8036,B 24.8049,C -3.221,E1 25.1487,E2 -291.3385} C_DIS
LIN {X 18.8401,Y 8.6363,Z 56,A 18.0556,B 24.8034,C -3.2328,E1 25.144,E2 -295.5954} C_DIS
LIN {X 18.0989,Y 10.0971,Z 56,A 22.6686,B 24.8019,C -3.2457,E1 25.1379,E2 -300.2145} C_DIS
LIN {X 17.1824,Y 11.5883,Z 56,A 27.501,B 24.8004,C -3.2577,E1 25.1306,E2 -305.0513} C_DIS
LIN {X 16.1542,Y 12.9835,Z 56,A 32.2543,B 24.799,C -3.2686,E1 25.1225,E2 -309.8078} C_DIS
LIN {X 15.0101,Y 14.2908,Z 56,A 37.0404,B 24.7978,C -3.2788,E1 25.1135,E2 -314.5971} C_DIS
LIN {X 13.7299,Y 15.5248,Z 56,A 41.9265,B 24.7966,C -3.2882,E1 25.1034,E2 -319.4855} C_DIS
LIN {X 12.4057,Y 16.6019,Z 56,A 46.6548,B 24.7956,C -3.2965,E1 25.093,E2 -324.2163} C_DIS
LIN {X 10.9794,Y 17.5777,Z 56,A 51.3848,B 24.7947,C -3.3034,E1 25.082,E2 -328.9472} C_DIS
LIN {X 9.4639,Y 18.4379,Z 56,A 56.2186,B 24.7939,C -3.3099,E1 25.0701,E2 -333.7824} C_DIS
LIN {X 7.8676,Y 19.1736,Z 56,A 60.8958,B 24.7934,C -3.3136,E1 25.0581,E2 -338.4571} C_DIS
LIN {X 6.3703,Y 19.7216,Z 56,A 65.453,B 24.7928,C -3.3184,E1 25.0461,E2 -343.0167} C_DIS
LIN {X 4.6788,Y 20.1899,Z 56,A 70.2628,B 24.7925,C -3.3208,E1 25.0331,E2 -347.8252} C_DIS
LIN {X 2.9949,Y 20.5075,Z 56,A 74.9908,B 24.7923,C -3.3223,E1 25.02,E2 -352.5517} C_DIS
LIN {X 1.2709,Y 20.6858,Z 56,A 79.7919,B 24.7923,C -3.3227,E1 25.0067,E2 -357.3512} C_DIS
LIN {X -0.46,Y 20.72,Z 56,A 84.5553,B 24.7924,C -3.3216,E1 24.9934,E2 -362.1118} C_DIS
LIN {X -2.1548,Y 20.6126,Z 56,A 89.3204,B 24.7926,C -3.3199,E1 24.9801,E2 -366.8752} C_DIS
LIN {X -3.8967,Y 20.3553,Z 56,A 94.192,B 24.7931,C -3.3164,E1 24.9667,E2 -371.7433} C_DIS
LIN {X -5.6456,Y 19.9411,Z 56,A 99.0777,B 24.7937,C -3.3112,E1 24.9536,E2 -376.6235} C_DIS
LIN {X -7.2363,Y 19.4203,Z 56,A 103.79,B 24.7944,C -3.306,E1 24.9412,E2 -381.3328} C_DIS
LIN {X -8.8612,Y 18.7353,Z 56,A 108.5563,B 24.7953,C -3.2984,E1 24.929,E2 -386.0924} C_DIS
LIN {X -10.239,Y 18.0193,Z 56,A 113.0452,B 24.7961,C -3.2923,E1 24.918,E2 -390.5794} C_DIS
LIN {X -11.7563,Y 17.0681,Z 56,A 117.9752,B 24.7973,C -3.283,E1 24.9065,E2 -395.5032} C_DIS
LIN {X -13.1479,Y 16.0207,Z 56,A 122.808,B 24.7985,C -3.2731,E1 24.8959,E2 -400.3302} C_DIS
LIN {X -14.464,Y 14.8434,Z 56,A 127.6385,B 24.7999,C -3.2618,E1 24.8861,E2 -405.1533} C_DIS
LIN {X -15.5924,Y 13.6528,Z 56,A 132.2799,B 24.8012,C -3.2513,E1 24.8774,E2 -409.7901} C_DIS
LIN {X -16.6815,Y 12.2985,Z 56,A 137.1615,B 24.8027,C -3.2392,E1 24.8691,E2 -414.666} C_DIS
LIN {X -17.6478,Y 10.8671,Z 56,A 141.9796,B 24.8042,C -3.2264,E1 24.8618,E2 -419.4777} C_DIS
LIN {X -18.512,Y 9.3182,Z 56,A 146.7863,B 24.806,C -3.2121,E1 24.8555,E2 -424.2757} C_DIS
LIN {X -19.1736,Y 7.8676,Z 56,A 151.1687,B 24.8075,C -3.1991,E1 24.8507,E2 -428.6511} C_DIS
LIN {X -19.7216,Y 6.3703,Z 56,A 155.7672,B 24.809,C -3.1866,E1 24.8465,E2 -433.2458} C_DIS
LIN {X -20.1899,Y 4.6788,Z 56,A 160.6442,B 24.8108,C -3.1718,E1 24.8432,E2 -438.116} C_DIS
LIN {X -20.5075,Y 2.9949,Z 56,A 165.3845,B 24.8126,C -3.1571,E1 24.841,E2 -442.8492} C_DIS
LIN {X -20.6858,Y 1.2709,Z 56,A 170.2217,B 24.8143,C -3.1424,E1 24.8399,E2 -447.6801} C_DIS
LIN {X -20.7189,Y -0.5147,Z 56,A 175.2425,B 24.8161,C -3.1273,E1 24.8399,E2 -452.6952} C_DIS
LIN {X -20.5986,Y -2.2843,Z 56,A 179.9885,B 24.818,C -3.1117,E1 24.8411,E2 -457.4321} C_DIS
LIN {X -20.3685,Y -3.8281,Z 56,A -175.4913,B 24.8194,C -3.0994,E1 24.8432,E2 -461.9497} C_DIS
LIN {X -19.974,Y -5.5276,Z 56,A -170.6418,B 24.8211,C -3.0852,E1 24.8466,E2 -466.7935} C_DIS
LIN {X -19.4261,Y -7.2209,Z 56,A -165.8138,B 24.8227,C -3.0707,E1 24.851,E2 -471.6143} C_DIS
LIN {X -18.8358,Y -8.6455,Z 56,A -161.3496,B 24.824,C -3.0598,E1 24.856,E2 -476.0769} C_DIS
LIN {X -18.0193,Y -10.239,Z 56,A -156.3699,B 24.8255,C -3.0469,E1 24.8626,E2 -481.052} C_DIS
LIN {X -17.0681,Y -11.7563,Z 56,A -151.4328,B 24.8269,C -3.0346,E1 24.8701,E2 -485.9844} C_DIS
LIN {X -16.0103,Y -13.1606,Z 56,A -146.5699,B 24.8282,C -3.0233,E1 24.8785,E2 -490.8434} C_DIS
LIN {X -14.8434,Y -14.464,Z 56,A -141.7685,B 24.8294,C -3.0129,E1 24.8877,E2 -495.6409} C_DIS
LIN {X -13.6528,Y -15.5924,Z 56,A -137.1326,B 24.8303,C -3.0047,E1 24.8972,E2 -500.2757} C_DIS
LIN {X -12.2985,Y -16.6815,Z 56,A -132.2609,B 24.8312,C -2.9967,E1 24.908,E2 -505.1462} C_DIS
LIN {X -10.8582,Y -17.6531,Z 56,A -127.4456,B 24.832,C -2.9896,E1 24.9193,E2 -509.96} C_DIS
LIN {X -9.3182,Y -18.512,Z 56,A -122.6677,B 24.8328,C -2.9829,E1 24.9311,E2 -514.7352} C_DIS
LIN {X -7.8676,Y -19.1736,Z 56,A -118.3049,B 24.8333,C -2.9781,E1 24.9423,E2 -519.0968} C_DIS
LIN {X -6.3703,Y -19.7216,Z 56,A -113.7304,B 24.8336,C -2.9756,E1 24.9544,E2 -523.6742} C_DIS
LIN {X -4.6788,Y -20.1899,Z 56,A -108.8821,B 24.8339,C -2.973,E1 24.9675,E2 -528.523} C_DIS
LIN {X -2.9944,Y -20.5076,Z 56,A -104.1726,B 24.8341,C -2.9714,E1 24.9805,E2 -533.2333} C_DIS
LIN {X -1.2709,Y -20.6858,Z 56,A -99.3709,B 24.8341,C -2.9714,E1 24.9938,E2 -538.0369} C_DIS
LIN {X 0.0545,Y -20.7204,Z 56,A -96.9596,B 24.835,C -2.9631,E1 25.0005,E2 -540.4289} C_DIS
Enddeposition()
LIN {X 0.0545,Y -20.7204,Z 56,A -96.9596,B 24.835,C -2.9631,E1 25.0005,E2 -540.4289} C_DIS
Startdeposition()
$VEL.CP = VEL_PRINT
LIN {X -0.0881,Y -19.7268,Z 56,A -98.5569,B 24.834,C -2.9724,E1 24.9961,E2 -538.8536} C_DIS
LIN {X -1.8243,Y -19.6424,Z 56,A -103.6074,B 24.834,C -2.9724,E1 24.982,E2 -533.8011} C_DIS
LIN {X -3.5089,Y -19.4123,Z 56,A -108.5479,B 24.8338,C -2.9737,E1 24.9684,E2 -528.8592} C_DIS
LIN {X -5.1546,Y -19.0416,Z 56,A -113.1931,B 24.8334,C -2.9777,E1 24.9558,E2 -524.2172} C_DIS
LIN {X -6.257,Y -18.7082,Z 56,A -116.5507,B 24.8331,C -2.9801,E1 24.9469,E2 -520.8593} C_DIS
LIN {X -7.683,Y -18.1693,Z 56,A -121.1962,B 24.8328,C -2.9831,E1 24.9348,E2 -516.2108} C_DIS
LIN {X -9.228,Y -17.4355,Z 56,A -126.2699,B 24.8321,C -2.9885,E1 24.9222,E2 -511.1365} C_DIS
LIN {X -10.6979,Y -16.5743,Z 56,A -131.1724,B 24.8313,C -2.9958,E1 24.9105,E2 -506.2362} C_DIS
LIN {X -12.0922,Y -15.5863,Z 56,A -136.2592,B 24.8304,C -3.0036,E1 24.8991,E2 -501.1498} C_DIS
LIN {X -13.7225,Y -14.1721,Z 56,A -143.0941,B 24.8293,C -3.0133,E1 24.8851,E2 -494.3104} C_DIS
LIN {X -15.0819,Y -12.7161,Z 56,A -148.3283,B 24.8276,C -3.0282,E1 24.8754,E2 -489.0884} C_DIS
LIN {X -16.1119,Y -11.3826,Z 56,A -153.234,B 24.8263,C -3.0397,E1 24.8673,E2 -484.1867} C_DIS
LIN {X -17.1598,Y -9.7316,Z 56,A -158.8779,B 24.8246,C -3.0543,E1 24.8591,E2 -478.5487} C_DIS
LIN {X -17.9368,Y -8.212,Z 56,A -164.0015,B 24.8232,C -3.0671,E1 24.8529,E2 -473.4281} C_DIS
LIN {X -18.6229,Y -6.5065,Z 56,A -169.2856,B 24.8214,C -3.0825,E1 24.8477,E2 -468.1509} C_DIS
LIN {X -19.1186,Y -4.8613,Z 56,A -174.3634,B 24.8197,C -3.0968,E1 24.8439,E2 -463.0781} C_DIS
LIN {X -19.4744,Y -3.1483,Z 56,A -179.4543,B 24.8179,C -3.1121,E1 24.8413,E2 -457.9937} C_DIS
LIN {X -19.6752,Y -1.4271,Z 56,A 175.4882,B 24.8161,C -3.1275,E1 24.84,E2 -452.9427} C_DIS
LIN {X -19.7219,Y 0.4555,Z 56,A 170.2092,B 24.814,C -3.1451,E1 24.84,E2 -447.6741} C_DIS
LIN {X -19.611,Y 2.134,Z 56,A 165.7014,B 24.812,C -3.1615,E1 24.8409,E2 -443.1786} C_DIS
LIN {X -19.4341,Y 3.3871,Z 56,A 161.3227,B 24.811,C -3.1707,E1 24.8428,E2 -438.7957} C_DIS
LIN {X -19.0589,Y 5.0896,Z 56,A 156.2338,B 24.8091,C -3.1861,E1 24.8462,E2 -433.7141} C_DIS
LIN {X -18.5341,Y 6.7554,Z 56,A 151.0593,B 24.8073,C -3.201,E1 24.8508,E2 -428.5458} C_DIS
LIN {X -17.8685,Y 8.3586,Z 56,A 145.8287,B 24.8056,C -3.2151,E1 24.8567,E2 -423.3203} C_DIS
LIN {X -17.1974,Y 9.6646,Z 56,A 141.1784,B 24.8043,C -3.2258,E1 24.863,E2 -418.6711} C_DIS
LIN {X -16.082,Y 11.4246,Z 56,A 135.7365,B 24.802,C -3.2443,E1 24.8714,E2 -413.2462} C_DIS
LIN {X -15.0202,Y 12.7882,Z 56,A 130.8725,B 24.8004,C -3.2576,E1 24.8799,E2 -408.3915} C_DIS
LIN {X -14.1301,Y 13.766,Z 56,A 126.7466,B 24.7994,C -3.2656,E1 24.8878,E2 -404.2669} C_DIS
LIN {X -12.8858,Y 14.9371,Z 56,A 121.8664,B 24.798,C -3.277,E1 24.8979,E2 -399.3944} C_DIS
LIN {X -11.5373,Y 16.0015,Z 56,A 116.7083,B 24.7968,C -3.2864,E1 24.9094,E2 -394.2403} C_DIS
LIN {X -10.0607,Y 16.9687,Z 56,A 111.6051,B 24.7957,C -3.2958,E1 24.9215,E2 -389.1434} C_DIS
LIN {X -8.5516,Y 17.777,Z 56,A 106.6395,B 24.7947,C -3.3037,E1 24.9338,E2 -384.1833} C_DIS
LIN {X -7.1071,Y 18.402,Z 56,A 102.6143,B 24.7936,C -3.3126,E1 24.9442,E2 -380.1703} C_DIS
LIN {X -6.1217,Y 18.7531,Z 56,A 99.567,B 24.7931,C -3.3162,E1 24.9522,E2 -377.1257} C_DIS
LIN {X -4.8505,Y 19.1214,Z 56,A 95.1538,B 24.793,C -3.3171,E1 24.9641,E2 -372.7077} C_DIS
LIN {X -3.2128,Y 19.4636,Z 56,A 90.2894,B 24.7925,C -3.3207,E1 24.9775,E2 -367.8469} C_DIS
LIN {X -1.4919,Y 19.6706,Z 56,A 85.2224,B 24.7922,C -3.323,E1 24.9915,E2 -362.7826} C_DIS
LIN {X 0.224,Y 19.7259,Z 56,A 80.1873,B 24.7922,C -3.3239,E1 25.0056,E2 -357.7494} C_DIS
LIN {X 2.3237,Y 19.5896,Z 56,A 74.6405,B 24.7917,C -3.3271,E1 25.021,E2 -352.2132} C_DIS
LIN {X 3.3345,Y 19.4432,Z 56,A 71.1493,B 24.7923,C -3.3227,E1 25.0306,E2 -348.7151} C_DIS
LIN {X 4.9587,Y 19.0936,Z 56,A 66.4427,B 24.7925,C -3.321,E1 25.0434,E2 -344.011} C_DIS
LIN {X 6.4676,Y 18.6364,Z 56,A 61.8864,B 24.7929,C -3.3176,E1 25.0555,E2 -339.4552} C_DIS
LIN {X 7.9982,Y 18.0332,Z 56,A 56.9887,B 24.7936,C -3.3119,E1 25.0681,E2 -334.5553} C_DIS
LIN {X 9.9673,Y 17.0238,Z 56,A 51.2761,B 24.794,C -3.3091,E1 25.0822,E2 -328.8522} C_DIS
LIN {X 10.9854,Y 16.3853,Z 56,A 46.5897,B 24.7958,C -3.2943,E1 25.0932,E2 -324.1461} C_DIS
LIN {X 12.705,Y 15.091,Z 56,A 41.4966,B 24.796,C -3.2926,E1 25.1043,E2 -319.068} C_DIS
LIN {X 13.5852,Y 14.304,Z 56,A 37.4234,B 24.7976,C -3.2806,E1 25.1127,E2 -314.9827} C_DIS
LIN {X 15.0177,Y 12.7914,Z 56,A 32.2328,B 24.7983,C -3.2749,E1 25.1225,E2 -309.8014} C_DIS
LIN {X 15.752,Y 11.8756,Z 56,A 28.0547,B 24.8001,C -3.2602,E1 25.1297,E2 -305.6083} C_DIS
LIN {X 16.7981,Y 10.343,Z 56,A 22.9571,B 24.8014,C -3.2494,E1 25.1375,E2 -300.5104} C_DIS
LIN {X 17.4999,Y 9.1052,Z 56,A 18.5989,B 24.803,C -3.2365,E1 25.1433,E2 -296.1445} C_DIS
LIN {X 18.2124,Y 7.5797,Z 56,A 13.7705,B 24.8046,C -3.2236,E1 25.1488,E2 -291.3116} C_DIS
LIN {X 18.7891,Y 6.0096,Z 56,A 8.9135,B 24.8063,C -3.2096,E1 25.1532,E2 -286.449} C_DIS
LIN {X 19.2356,Y 4.3746,Z 56,A 4.0103,B 24.808,C -3.1952,E1 25.1565,E2 -281.5399} C_DIS
LIN {X 19.5522,Y 2.6197,Z 56,A -0.9965,B 24.8097,C -3.1811,E1 25.1587,E2 -276.5291} C_DIS
LIN {X 19.6699,Y 1.5001,Z 56,A -4.4216,B 24.8111,C -3.1695,E1 25.1595,E2 -273.0968} C_DIS
LIN {X 19.7262,Y -0.2286,Z 56,A -9.4909,B 24.813,C -3.1535,E1 25.1597,E2 -268.0196} C_DIS
LIN {X 19.6629,Y -1.5886,Z 56,A -12.9781,B 24.8139,C -3.1456,E1 25.159,E2 -264.5345} C_DIS
LIN {X 19.4851,Y -3.08,Z 56,A -17.5606,B 24.8158,C -3.1299,E1 25.1573,E2 -259.9419} C_DIS
LIN {X 19.1697,Y -4.6555,Z 56,A -22.2938,B 24.8176,C -3.1149,E1 25.1544,E2 -255.2006} C_DIS
LIN {X 18.6986,Y -6.286,Z 56,A -27.3015,B 24.8194,C -3.0992,E1 25.1502,E2 -250.1842} C_DIS
LIN {X 18.0472,Y -7.9661,Z 56,A -32.2339,B 24.8209,C -3.0865,E1 25.145,E2 -245.2489} C_DIS
LIN {X 16.9468,Y -10.0977,Z 56,A -40.4243,B 24.8245,C -3.0556,E1 25.1339,E2 -237.028} C_DIS
LIN {X 15.6846,Y -11.9647,Z 56,A -45.8265,B 24.8253,C -3.0485,E1 25.125,E2 -231.6351} C_DIS
LIN {X 14.5698,Y -13.2994,Z 56,A -50.3198,B 24.8262,C -3.0409,E1 25.1168,E2 -227.144} C_DIS
LIN {X 13.691,Y -14.2024,Z 56,A -54.3207,B 24.8275,C -3.0293,E1 25.1089,E2 -223.1324} C_DIS
LIN {X 12.4733,Y -15.283,Z 56,A -59.1818,B 24.8288,C -3.0178,E1 25.0986,E2 -218.263} C_DIS
LIN {X 11.0853,Y -16.3178,Z 56,A -64.2082,B 24.83,C -3.0078,E1 25.0871,E2 -213.2305} C_DIS
LIN {X 9.6761,Y -17.191,Z 56,A -69.2523,B 24.8311,C -2.9974,E1 25.075,E2 -208.177} C_DIS
LIN {X 8.1972,Y -17.9434,Z 56,A -73.5733,B 24.8315,C -2.9938,E1 25.0641,E2 -203.8589} C_DIS
LIN {X 6.7993,Y -18.5182,Z 56,A -78.0501,B 24.8323,C -2.9873,E1 25.0524,E2 -199.3764} C_DIS
LIN {X 5.142,Y -19.045,Z 56,A -82.9286,B 24.8328,C -2.983,E1 25.0394,E2 -194.4962} C_DIS
LIN {X 4.0953,Y -19.2974,Z 56,A -86.3765,B 24.8333,C -2.9779,E1 25.03,E2 -191.0407} C_DIS
LIN {X 2.3765,Y -19.5834,Z 56,A -91.2927,B 24.8336,C -2.9755,E1 25.0164,E2 -186.1232} C_DIS
LIN {X 0.7228,Y -19.7136,Z 56,A -96.1174,B 24.8338,C -2.9735,E1 25.0029,E2 -181.2957} C_DIS
LIN {X 0.7228,Y -19.7136,Z 56,A -96.1174,B 24.8338,C -2.9735,E1 25.0029,E2 -181.2957} C_DIS
Enddeposition()
LIN {X 0.0479,Y -18.7257,Z 56,A -97.6494,B 24.8316,C -2.9934,E1 24.9988,E2 -179.8111} C_DIS
Startdeposition()
$VEL.CP = VEL_PRINT
LIN {X 1.0717,Y -18.6983,Z 56,A -92.5355,B 24.83,C -3.0073,E1 25.0131,E2 -184.957} C_DIS
LIN {X 2.7757,Y -18.5223,Z 56,A -87.3343,B 24.8297,C -3.0103,E1 25.0275,E2 -190.1611} C_DIS
LIN {X 5.0425,Y -18.0372,Z 56,A -79.3132,B 24.8281,C -3.0239,E1 25.0493,E2 -198.2029} C_DIS
LIN {X 6.9904,Y -17.3756,Z 56,A -74.3167,B 24.8283,C -3.0222,E1 25.0624,E2 -203.1846} C_DIS
LIN {X 7.9045,Y -16.9792,Z 56,A -71.136,B 24.8277,C -3.0278,E1 25.0705,E2 -206.3706} C_DIS
LIN {X 9.1416,Y -16.3464,Z 56,A -67.0853,B 24.8271,C -3.0332,E1 25.0804,E2 -210.4229} C_DIS
LIN {X 10.1769,Y -15.7226,Z 56,A -63.5066,B 24.8264,C -3.0391,E1 25.0889,E2 -214.004} C_DIS
LIN {X 11.0514,Y -15.1209,Z 56,A -60.1871,B 24.8256,C -3.0461,E1 25.0965,E2 -217.3287} C_DIS
LIN {X 11.9964,Y -14.3822,Z 56,A -56.2602,B 24.8244,C -3.0561,E1 25.105,E2 -221.2644} C_DIS
LIN {X 12.9802,Y -13.5014,Z 56,A -52.1323,B 24.8233,C -3.0661,E1 25.1135,E2 -225.3992} C_DIS
LIN {X 14.2616,Y -12.14,Z 56,A -46.1636,B 24.8214,C -3.0824,E1 25.1246,E2 -231.38} C_DIS
LIN {X 15.217,Y -10.9188,Z 56,A -42.1601,B 24.8207,C -3.0883,E1 25.1313,E2 -235.3782} C_DIS
LIN {X 16.0802,Y -9.6019,Z 56,A -36.2015,B 24.8179,C -3.1119,E1 25.1401,E2 -241.3627} C_DIS
LIN {X 17.0238,Y -7.8088,Z 56,A -31.1864,B 24.8171,C -3.1189,E1 25.1463,E2 -246.3675} C_DIS
LIN {X 17.3929,Y -6.9474,Z 56,A -28.148,B 24.8159,C -3.129,E1 25.1495,E2 -249.4131} C_DIS
LIN {X 17.9439,Y -5.366,Z 56,A -22.8775,B 24.8139,C -3.1459,E1 25.1541,E2 -254.6937} C_DIS
LIN {X 18.3528,Y -3.7345,Z 56,A -17.7579,B 24.8121,C -3.1615,E1 25.1572,E2 -259.8205} C_DIS
LIN {X 18.6132,Y -2.079,Z 56,A -12.9086,B 24.8105,C -3.1748,E1 25.1591,E2 -264.6729} C_DIS
LIN {X 18.7201,Y -0.5775,Z 56,A -8.088,B 24.8085,C -3.1912,E1 25.1598,E2 -269.5036} C_DIS
LIN {X 18.7046,Y 0.9528,Z 56,A -3.4019,B 24.8067,C -3.2058,E1 25.1593,E2 -274.1964} C_DIS
LIN {X 18.5679,Y 2.4503,Z 56,A 0.8606,B 24.8054,C -3.2167,E1 25.158,E2 -278.4596} C_DIS
LIN {X 18.288,Y 4.0404,Z 56,A 6.0977,B 24.8032,C -3.2344,E1 25.1552,E2 -283.708} C_DIS
LIN {X 17.8444,Y 5.6872,Z 56,A 11.2411,B 24.8015,C -3.2489,E1 25.1511,E2 -288.8566} C_DIS
LIN {X 17.2777,Y 7.2283,Z 56,A 16.1872,B 24.7998,C -3.2624,E1 25.1461,E2 -293.8071} C_DIS
LIN {X 16.6222,Y 8.63,Z 56,A 20.5788,B 24.7986,C -3.2721,E1 25.1407,E2 -298.1983} C_DIS
LIN {X 16.1679,Y 9.4541,Z 56,A 24.304,B 24.7967,C -3.287,E1 25.1354,E2 -301.9397} C_DIS
LIN {X 14.7242,Y 11.5747,Z 56,A 30.8598,B 24.7958,C -3.2948,E1 25.1248,E2 -308.482} C_DIS
LIN {X 13.9583,Y 12.4876,Z 56,A 35.5686,B 24.7937,C -3.3118,E1 25.1162,E2 -313.21} C_DIS
LIN {X 12.6057,Y 13.8519,Z 56,A 40.4658,B 24.7932,C -3.3156,E1 25.1064,E2 -318.0957} C_DIS
LIN {X 11.6677,Y 14.6502,Z 56,A 45.323,B 24.7912,C -3.3312,E1 25.0958,E2 -322.9716} C_DIS
LIN {X 9.7909,Y 15.966,Z 56,A 51.3251,B 24.7908,C -3.3342,E1 25.0819,E2 -328.9609} C_DIS
LIN {X 8.5959,Y 16.64,Z 56,A 55.3848,B 24.7903,C -3.3388,E1 25.072,E2 -333.0196} C_DIS
LIN {X 7.4217,Y 17.1955,Z 56,A 59.987,B 24.7891,C -3.3477,E1 25.0603,E2 -337.6317} C_DIS
LIN {X 5.8866,Y 17.7796,Z 56,A 64.9745,B 24.7886,C -3.3518,E1 25.0471,E2 -342.6187} C_DIS
LIN {X 4.2976,Y 18.2294,Z 56,A 70.0403,B 24.7882,C -3.3548,E1 25.0334,E2 -347.6839} C_DIS
LIN {X 2.9768,Y 18.4908,Z 56,A 73.5366,B 24.7886,C -3.3523,E1 25.0239,E2 -351.1703} C_DIS
LIN {X 2.0441,Y 18.617,Z 56,A 76.5393,B 24.7884,C -3.3536,E1 25.0155,E2 -354.1738} C_DIS
LIN {X 0.5237,Y 18.7216,Z 56,A 82.4175,B 24.7875,C -3.3608,E1 24.9991,E2 -360.0675} C_DIS
LIN {X -1.5948,Y 18.6608,Z 56,A 88.242,B 24.7883,C -3.3545,E1 24.9829,E2 -365.8787} C_DIS
LIN {X -3.2831,Y 18.4389,Z 56,A 93.3767,B 24.7888,C -3.3507,E1 24.9688,E2 -371.0087} C_DIS
LIN {X -4.8957,Y 18.0778,Z 56,A 97.9028,B 24.7897,C -3.3432,E1 24.9565,E2 -375.5233} C_DIS
LIN {X -6.3576,Y 17.6169,Z 56,A 103.4767,B 24.7898,C -3.3422,E1 24.9417,E2 -381.1051} C_DIS
LIN {X -7.8009,Y 17.0273,Z 56,A 107.8698,B 24.7909,C -3.3336,E1 24.9305,E2 -385.4881} C_DIS
LIN {X -9.0833,Y 16.3784,Z 56,A 111.8588,B 24.792,C -3.3246,E1 24.9207,E2 -389.4668} C_DIS
LIN {X -10.0157,Y 15.826,Z 56,A 115.5191,B 24.7926,C -3.3202,E1 24.912,E2 -393.1278} C_DIS
LIN {X -10.8133,Y 15.292,Z 56,A 118.6363,B 24.7932,C -3.3153,E1 24.9049,E2 -396.244} C_DIS
LIN {X -12.2209,Y 14.1925,Z 56,A 124.4961,B 24.7945,C -3.3053,E1 24.8922,E2 -402.1021} C_DIS
LIN {X -13.5687,Y 12.9101,Z 56,A 129.2453,B 24.7966,C -3.2884,E1 24.8829,E2 -406.8309} C_DIS
LIN {X -14.344,Y 12.0426,Z 56,A 133.1915,B 24.7975,C -3.281,E1 24.8756,E2 -410.7773} C_DIS
LIN {X -15.0592,Y 11.1356,Z 56,A 136.5513,B 24.7987,C -3.2713,E1 24.87,E2 -414.1297} C_DIS
LIN {X -15.7638,Y 10.1132,Z 56,A 140.7006,B 24.7998,C -3.2623,E1 24.8635,E2 -418.2781} C_DIS
LIN {X -16.407,Y 9.0328,Z 56,A 144.2263,B 24.8013,C -3.2504,E1 24.8587,E2 -421.7939} C_DIS
LIN {X -17.1295,Y 7.573,Z 56,A 150.5429,B 24.8025,C -3.2404,E1 24.8512,E2 -428.1209} C_DIS
LIN {X -17.9105,Y 5.4756,Z 56,A 156.3857,B 24.8054,C -3.2166,E1 24.846,E2 -433.94} C_DIS
LIN {X -18.2115,Y 4.3719,Z 56,A 160.3124,B 24.8065,C -3.2072,E1 24.8433,E2 -437.8671} C_DIS
LIN {X -18.6008,Y 2.1842,Z 56,A 167.1551,B 24.8091,C -3.1863,E1 24.8405,E2 -444.7004} C_DIS
LIN {X -18.7202,Y 0.5717,Z 56,A 171.8767,B 24.811,C -3.1702,E1 24.8398,E2 -449.4118} C_DIS
LIN {X -18.7071,Y -0.8997,Z 56,A 176.6211,B 24.8126,C -3.157,E1 24.8402,E2 -454.1532} C_DIS
LIN {X -18.5376,Y -2.6704,Z 56,A -177.9615,B 24.8146,C -3.1403,E1 24.842,E2 -459.5629} C_DIS
LIN {X -18.2327,Y -4.2836,Z 56,A -172.9037,B 24.8163,C -3.1253,E1 24.8449,E2 -464.6146} C_DIS
LIN {X -17.7999,Y -5.8255,Z 56,A -168.5719,B 24.8182,C -3.1092,E1 24.8484,E2 -468.9328} C_DIS
LIN {X -17.366,Y -7.0141,Z 56,A -164.127,B 24.8193,C -3.1002,E1 24.8528,E2 -473.3812} C_DIS
LIN {X -16.7415,Y -8.3944,Z 56,A -159.1407,B 24.8206,C -3.0889,E1 24.8589,E2 -478.3674} C_DIS
LIN {X -15.579,Y -10.3958,Z 56,A -152.261,B 24.8228,C -3.0702,E1 24.8689,E2 -485.2375} C_DIS
LIN {X -14.5642,Y -11.7754,Z 56,A -147.6154,B 24.8245,C -3.0557,E1 24.8768,E2 -489.8704} C_DIS
LIN {X -13.8489,Y -12.6085,Z 56,A -144.1751,B 24.8253,C -3.0486,E1 24.8831,E2 -493.3094} C_DIS
LIN {X -13.0417,Y -13.4422,Z 56,A -140.4102,B 24.826,C -3.0423,E1 24.8906,E2 -497.0751} C_DIS
LIN {X -11.7655,Y -14.5721,Z 56,A -134.0418,B 24.8265,C -3.0379,E1 24.9042,E2 -503.4574} C_DIS
LIN {X -9.9916,Y -15.8412,Z 56,A -128.1403,B 24.8281,C -3.0239,E1 24.9178,E2 -509.345} C_DIS
LIN {X -8.5345,Y -16.6714,Z 56,A -122.9954,B 24.8289,C -3.0174,E1 24.9305,E2 -514.4889} C_DIS
LIN {X -6.9741,Y -17.3822,Z 56,A -118.1756,B 24.8297,C -3.0097,E1 24.9428,E2 -519.3018} C_DIS
LIN {X -5.9944,Y -17.7436,Z 56,A -114.5594,B 24.8297,C -3.0095,E1 24.9524,E2 -522.9243} C_DIS
LIN {X -4.5488,Y -18.1685,Z 56,A -110.6667,B 24.8305,C -3.0026,E1 24.9628,E2 -526.8068} C_DIS
LIN {X -3.1101,Y -18.4689,Z 56,A -105.4066,B 24.8302,C -3.0054,E1 24.9773,E2 -532.0794} C_DIS
LIN {X -1.4631,Y -18.6718,Z 56,A -100.2805,B 24.8302,C -3.0054,E1 24.9915,E2 -537.2081} C_DIS
LIN {X 0.0479,Y -18.7257,Z 56,A -97.6493,B 24.8316,C -2.9933,E1 24.9988,E2 -539.8111} C_DIS
Enddeposition()
LIN {X 0.0479,Y -18.7257,Z 56,A -97.6493,B 24.8316,C -2.9933,E1 24.9988,E2 -539.8111} C_DIS
Startdeposition()
$VEL.CP = VEL_PRINT
LIN {X -0.6251,Y -17.7199,Z 56,A -100.4629,B 24.8301,C -3.0067,E1 24.991,E2 -537.029} C_DIS
LIN {X -2.3598,Y -17.5733,Z 56,A -105.5447,B 24.8297,C -3.0103,E1 24.9769,E2 -531.9528} C_DIS
LIN {X -3.3384,Y -17.4138,Z 56,A -109.0436,B 24.8297,C -3.0098,E1 24.9673,E2 -528.4491} C_DIS
LIN {X -4.7978,Y -17.0692,Z 56,A -113.7537,B 24.8294,C -3.0131,E1 24.9545,E2 -523.7402} C_DIS
LIN {X -5.9593,Y -16.6991,Z 56,A -118.0705,B 24.8292,C -3.0144,E1 24.9431,E2 -519.4181} C_DIS
LIN {X -7.1429,Y -16.2287,Z 56,A -122.2581,B 24.8288,C -3.0182,E1 24.9323,E2 -515.2299} C_DIS
LIN {X -8.6063,Y -15.5023,Z 56,A -127.531,B 24.828,C -3.0248,E1 24.9193,E2 -509.9583} C_DIS
LIN {X -9.8968,Y -14.7119,Z 56,A -133.4934,B 24.8277,C -3.0278,E1 24.9054,E2 -503.9837} C_DIS
LIN {X -12.2878,Y -12.7827,Z 56,A -142.7872,B 24.8253,C -3.0488,E1 24.8858,E2 -494.7036} C_DIS
LIN {X -13.57,Y -11.4128,Z 56,A -148.4206,B 24.8236,C -3.0634,E1 24.8754,E2 -489.0801} C_DIS
LIN {X -14.5178,Y -10.1797,Z 56,A -153.0121,B 24.822,C -3.0768,E1 24.8678,E2 -484.4984} C_DIS
LIN {X -15.4916,Y -8.6242,Z 56,A -160.0465,B 24.8207,C -3.0885,E1 24.8577,E2 -477.4558} C_DIS
LIN {X -16.4923,Y -6.5078,Z 56,A -168.1549,B 24.8184,C -3.108,E1 24.8488,E2 -469.3493} C_DIS
LIN {X -17.0311,Y -4.932,Z 56,A -173.4214,B 24.8165,C -3.124,E1 24.8446,E2 -464.0907} C_DIS
LIN {X -17.5169,Y -2.747,Z 56,A -179.9612,B 24.8137,C -3.1475,E1 24.8412,E2 -457.5687} C_DIS
LIN {X -17.7107,Y -0.8441,Z 56,A 174.6001,B 24.8112,C -3.1685,E1 24.8399,E2 -452.1475} C_DIS
LIN {X -17.7219,Y 0.5629,Z 56,A 169.4891,B 24.8097,C -3.1811,E1 24.8399,E2 -447.0361} C_DIS
LIN {X -17.6291,Y 1.8961,Z 56,A 165.1034,B 24.8081,C -3.1944,E1 24.8411,E2 -442.6558} C_DIS
LIN {X -17.4274,Y 3.2683,Z 56,A 160.4089,B 24.8065,C -3.2077,E1 24.8433,E2 -437.9654} C_DIS
LIN {X -17.1166,Y 4.6271,Z 56,A 155.8857,B 24.8048,C -3.2215,E1 24.8464,E2 -433.4487} C_DIS
LIN {X -16.6756,Y 6.0259,Z 56,A 151.4745,B 24.803,C -3.2366,E1 24.8503,E2 -429.0486} C_DIS
LIN {X -16.1806,Y 7.2511,Z 56,A 147.0486,B 24.8015,C -3.2487,E1 24.8551,E2 -424.6271} C_DIS
LIN {X -15.4276,Y 8.7391,Z 56,A 140.9114,B 24.7999,C -3.2619,E1 24.8632,E2 -418.4891} C_DIS
LIN {X -14.5437,Y 10.1424,Z 56,A 135.4379,B 24.7981,C -3.2759,E1 24.8718,E2 -413.022} C_DIS
LIN {X -13.1232,Y 11.9237,Z 56,A 128.7084,B 24.7956,C -3.2963,E1 24.8839,E2 -406.3104} C_DIS
LIN {X -11.9855,Y 13.0664,Z 56,A 123.3254,B 24.7942,C -3.3076,E1 24.8947,E2 -400.9324} C_DIS
LIN {X -10.7201,Y 14.1236,Z 56,A 117.8889,B 24.7928,C -3.3184,E1 24.9065,E2 -395.5013} C_DIS
LIN {X -9.3043,Y 15.094,Z 56,A 113.0275,B 24.7912,C -3.3313,E1 24.9178,E2 -390.6548} C_DIS
LIN {X -8.172,Y 15.7355,Z 56,A 108.767,B 24.7904,C -3.3381,E1 24.9283,E2 -386.3984} C_DIS
LIN {X -7.0519,Y 16.2682,Z 56,A 103.7108,B 24.7902,C -3.3395,E1 24.9412,E2 -381.3334} C_DIS
LIN {X -4.9345,Y 17.0303,Z 56,A 97.2954,B 24.7886,C -3.3518,E1 24.9581,E2 -374.9354} C_DIS
LIN {X -3.2844,Y 17.424,Z 56,A 91.4538,B 24.7882,C -3.3548,E1 24.974,E2 -369.0936} C_DIS
LIN {X -1.8458,Y 17.633,Z 56,A 87.9673,B 24.7871,C -3.3638,E1 24.9836,E2 -365.6259} C_DIS
LIN {X -1.0386,Y 17.7005,Z 56,A 84.4988,B 24.7875,C -3.3603,E1 24.9933,E2 -362.1479} C_DIS
LIN {X 0.1791,Y 17.7302,Z 56,A 80.3697,B 24.7875,C -3.3601,E1 25.0048,E2 -358.0182} C_DIS
LIN {X 1.5699,Y 17.6613,Z 56,A 75.7551,B 24.7877,C -3.3594,E1 25.0177,E2 -353.4039} C_DIS
LIN {X 2.9396,Y 17.4855,Z 56,A 71.1135,B 24.7879,C -3.3571,E1 25.0305,E2 -348.7613} C_DIS
LIN {X 4.5788,Y 17.1294,Z 56,A 65.7854,B 24.7882,C -3.3548,E1 25.0449,E2 -343.4353} C_DIS
LIN {X 6.0876,Y 16.6532,Z 56,A 60.2462,B 24.7891,C -3.3478,E1 25.0596,E2 -337.8904} C_DIS
LIN {X 8.4762,Y 15.5736,Z 56,A 51.4194,B 24.7907,C -3.3353,E1 25.0817,E2 -329.0574} C_DIS
LIN {X 10.0903,Y 14.5798,Z 56,A 46.3497,B 24.7909,C -3.3334,E1 25.0935,E2 -324} C_DIS
LIN {X 11.0363,Y 13.8773,Z 56,A 42.4484,B 24.7919,C -3.3261,E1 25.1021,E2 -320.0956} C_DIS
LIN {X 12.2301,Y 12.8381,Z 56,A 37.0888,B 24.7933,C -3.3143,E1 25.1132,E2 -314.7295} C_DIS
LIN {X 13.1943,Y 11.8448,Z 56,A 33.3523,B 24.7938,C -3.3105,E1 25.1203,E2 -311.0004} C_DIS
LIN {X 14.0619,Y 10.8005,Z 56,A 28.2417,B 24.7958,C -3.2946,E1 25.1293,E2 -305.8759} C_DIS
LIN {X 14.9002,Y 9.6112,Z 56,A 24.131,B 24.7966,C -3.2879,E1 25.1357,E2 -301.7695} C_DIS
LIN {X 15.5206,Y 8.573,Z 56,A 19.9058,B 24.7982,C -3.2751,E1 25.1415,E2 -297.5359} C_DIS
LIN {X 16.0252,Y 7.5888,Z 56,A 16.2541,B 24.7995,C -3.2647,E1 25.146,E2 -293.8792} C_DIS
LIN {X 16.6578,Y 6.0749,Z 56,A 11.0048,B 24.8013,C -3.2503,E1 25.1513,E2 -288.6247} C_DIS
LIN {X 17.1355,Y 4.5558,Z 56,A 5.8849,B 24.8031,C -3.2354,E1 25.1553,E2 -283.499} C_DIS
LIN {X 17.4936,Y 2.8918,Z 56,A 0.9051,B 24.8046,C -3.2234,E1 25.158,E2 -278.5197} C_DIS
LIN {X 17.685,Y 1.2753,Z 56,A -5.066,B 24.8073,C -3.201,E1 25.1596,E2 -272.5309} C_DIS
LIN {X 17.7287,Y -0.2918,Z 56,A -9.8876,B 24.8089,C -3.1874,E1 25.1596,E2 -267.7057} C_DIS
LIN {X 17.6195,Y -1.9854,Z 56,A -15.2275,B 24.8108,C -3.1716,E1 25.1583,E2 -262.3599} C_DIS
LIN {X 17.373,Y -3.5445,Z 56,A -20.3716,B 24.8128,C -3.1554,E1 25.1558,E2 -257.2076} C_DIS
LIN {X 16.9436,Y -5.2248,Z 56,A -26.1266,B 24.815,C -3.137,E1 25.1514,E2 -251.4419} C_DIS
LIN {X 16.4058,Y -6.726,Z 56,A -30.7374,B 24.8162,C -3.1263,E1 25.1468,E2 -246.8316} C_DIS
LIN {X 15.8101,Y -8.0264,Z 56,A -34.6901,B 24.8171,C -3.1187,E1 25.1421,E2 -242.8821} C_DIS
LIN {X 15.2496,Y -9.0457,Z 56,A -38.8367,B 24.8188,C -3.1047,E1 25.1364,E2 -238.724} C_DIS
LIN {X 14.4912,Y -10.2169,Z 56,A -44.391,B 24.8212,C -3.0838,E1 25.1276,E2 -233.1474} C_DIS
LIN {X 13.1046,Y -11.944,Z 56,A -51.1073,B 24.8229,C -3.0694,E1 25.1155,E2 -226.4276} C_DIS
LIN {X 12.1228,Y -12.9393,Z 56,A -55.4813,B 24.824,C -3.0601,E1 25.1067,E2 -222.0497} C_DIS
LIN {X 10.9912,Y -13.9133,Z 56,A -60.1041,B 24.825,C -3.0513,E1 25.0967,E2 -217.4237} C_DIS
LIN {X 9.9954,Y -14.6451,Z 56,A -64.7779,B 24.8265,C -3.0383,E1 25.086,E2 -212.7349} C_DIS
LIN {X 8.1925,Y -15.7248,Z 56,A -70.7032,B 24.8271,C -3.033,E1 25.0716,E2 -206.8146} C_DIS
LIN {X 7.0464,Y -16.2706,Z 56,A -75.3892,B 24.8283,C -3.0227,E1 25.0596,E2 -202.1158} C_DIS
LIN {X 5.5735,Y -16.832,Z 56,A -80.3617,B 24.8289,C -3.0172,E1 25.0465,E2 -197.1403} C_DIS
LIN {X 3.6923,Y -17.3425,Z 56,A -85.7881,B 24.8289,C -3.0169,E1 25.0318,E2 -191.7213} C_DIS
LIN {X 2.5467,Y -17.5472,Z 56,A -90.1601,B 24.8297,C -3.0103,E1 25.0197,E2 -187.3378} C_DIS
LIN {X 0.9797,Y -17.7039,Z 56,A -95.2399,B 24.8299,C -3.0079,E1 25.0056,E2 -182.2551} C_DIS
LIN {X 0.9797,Y -17.7039,Z 56,A -95.2399,B 24.8299,C -3.0079,E1 25.0056,E2 -182.2551} C_DIS
Enddeposition()
LIN {X 0.0625,Y -16.7275,Z 56,A -97.2929,B 24.8274,C -3.03,E1 25,E2 -180.2549} C_DIS
Startdeposition()
$VEL.CP = VEL_PRINT
LIN {X 1.2327,Y -16.6875,Z 56,A -91.7228,B 24.8262,C -3.0407,E1 25.0156,E2 -185.8485} C_DIS
LIN {X 3.1344,Y -16.4368,Z 56,A -84.6016,B 24.8253,C -3.0489,E1 25.0353,E2 -192.9823} C_DIS
LIN {X 4.7943,Y -16.0315,Z 56,A -78.7167,B 24.8245,C -3.0553,E1 25.0511,E2 -198.8727} C_DIS
LIN {X 6.8786,Y -15.2534,Z 56,A -72.0427,B 24.8241,C -3.0591,E1 25.0684,E2 -205.5407} C_DIS
LIN {X 8.5247,Y -14.3986,Z 56,A -64.7554,B 24.822,C -3.0767,E1 25.0862,E2 -212.8487} C_DIS
LIN {X 9.8789,Y -13.5052,Z 56,A -59.7733,B 24.8213,C -3.0833,E1 25.0976,E2 -217.8291} C_DIS
LIN {X 11.0022,Y -12.6073,Z 56,A -55.2838,B 24.8204,C -3.0906,E1 25.1072,E2 -222.3187} C_DIS
LIN {X 11.9565,Y -11.7061,Z 56,A -50.7676,B 24.8192,C -3.1012,E1 25.1163,E2 -226.8413} C_DIS
LIN {X 12.917,Y -10.6371,Z 56,A -46.4562,B 24.8183,C -3.1085,E1 25.1242,E2 -231.1506} C_DIS
LIN {X 13.6817,Y -9.6336,Z 56,A -40.5301,B 24.8154,C -3.1332,E1 25.134,E2 -237.1067} C_DIS
LIN {X 14.7186,Y -7.9595,Z 56,A -35.313,B 24.8147,C -3.1392,E1 25.1413,E2 -242.3112} C_DIS
LIN {X 15.2213,Y -6.9506,Z 56,A -30.6719,B 24.8126,C -3.1571,E1 25.1469,E2 -246.9695} C_DIS
LIN {X 15.7327,Y -5.6987,Z 56,A -26.4467,B 24.8113,C -3.1674,E1 25.1512,E2 -251.1957} C_DIS
LIN {X 16.1141,Y -4.5071,Z 56,A -21.4013,B 24.809,C -3.187,E1 25.1552,E2 -256.2589} C_DIS
LIN {X 16.5161,Y -2.6864,Z 56,A -15.4551,B 24.8071,C -3.2029,E1 25.1583,E2 -262.2081} C_DIS
LIN {X 16.698,Y -1.0805,Z 56,A -10.3404,B 24.8054,C -3.2165,E1 25.1596,E2 -267.3246} C_DIS
LIN {X 16.7287,Y 0.3849,Z 56,A -5.6141,B 24.8038,C -3.2296,E1 25.1596,E2 -272.0538} C_DIS
LIN {X 16.6688,Y 1.4628,Z 56,A -1.577,B 24.8021,C -3.2439,E1 25.1589,E2 -276.101} C_DIS
LIN {X 16.5005,Y 2.7799,Z 56,A 3.1109,B 24.8002,C -3.259,E1 25.1569,E2 -280.797} C_DIS
LIN {X 16.1965,Y 4.2035,Z 56,A 7.4743,B 24.799,C -3.2685,E1 25.1542,E2 -285.1577} C_DIS
LIN {X 15.8579,Y 5.3404,Z 56,A 12.2144,B 24.7969,C -3.2861,E1 25.1502,E2 -289.9125} C_DIS
LIN {X 15.2655,Y 6.8526,Z 56,A 16.8812,B 24.7959,C -3.2941,E1 25.1452,E2 -294.5727} C_DIS
LIN {X 14.7551,Y 7.8923,Z 56,A 21.8969,B 24.7935,C -3.3134,E1 25.1388,E2 -299.6074} C_DIS
LIN {X 13.8549,Y 9.382,Z 56,A 28.2883,B 24.7912,C -3.3317,E1 25.129,E2 -306.0104} C_DIS
LIN {X 12.3237,Y 11.3189,Z 56,A 35.5931,B 24.7899,C -3.3417,E1 25.116,E2 -313.3054} C_DIS
LIN {X 11.351,Y 12.2944,Z 56,A 40.4161,B 24.7886,C -3.3521,E1 25.1063,E2 -318.1329} C_DIS
LIN {X 10.2023,Y 13.263,Z 56,A 46.1139,B 24.7869,C -3.3653,E1 25.0939,E2 -323.8408} C_DIS
LIN {X 8.9445,Y 14.1416,Z 56,A 51.8638,B 24.7854,C -3.3769,E1 25.0804,E2 -329.5993} C_DIS
LIN {X 6.8202,Y 15.2801,Z 56,A 59.343,B 24.7848,C -3.3815,E1 25.0617,E2 -337.0696} C_DIS
LIN {X 5.0086,Y 15.9657,Z 56,A 65.9212,B 24.7842,C -3.3868,E1 25.0444,E2 -343.647} C_DIS
LIN {X 3.9449,Y 16.2614,Z 56,A 70.1895,B 24.7835,C -3.3919,E1 25.0328,E2 -347.9212} C_DIS
LIN {X 2.0561,Y 16.6064,Z 56,A 76.5198,B 24.7835,C -3.3922,E1 25.0153,E2 -354.2464} C_DIS
LIN {X 0.0386,Y 16.7329,Z 56,A 82.3656,B 24.7843,C -3.3859,E1 24.9991,E2 -360.0755} C_DIS
LIN {X -0.9797,Y 16.7043,Z 56,A 86.4677,B 24.784,C -3.388,E1 24.9876,E2 -364.1834} C_DIS
LIN {X -2.3041,Y 16.5737,Z 56,A 90.7012,B 24.7845,C -3.3839,E1 24.9759,E2 -368.4098} C_DIS
LIN {X -3.5182,Y 16.3591,Z 56,A 95.502,B 24.7846,C -3.3833,E1 24.9627,E2 -373.2145} C_DIS
LIN {X -4.6408,Y 16.0764,Z 56,A 99.2657,B 24.7852,C -3.3784,E1 24.9526,E2 -376.9724} C_DIS
LIN {X -6.1334,Y 15.5684,Z 56,A 105.1432,B 24.7858,C -3.3736,E1 24.9372,E2 -382.8506} C_DIS
LIN {X -7.8692,Y 14.7673,Z 56,A 111.4901,B 24.7872,C -3.3627,E1 24.9214,E2 -389.188} C_DIS
LIN {X -9.1562,Y 14.0036,Z 56,A 115.967,B 24.7887,C -3.3511,E1 24.9108,E2 -393.6512} C_DIS
LIN {X -10.3424,Y 13.1541,Z 56,A 121.0903,B 24.7899,C -3.3415,E1 24.8993,E2 -398.7698} C_DIS
LIN {X -10.9847,Y 12.6227,Z 56,A 124.2949,B 24.7905,C -3.3365,E1 24.8925,E2 -401.9748} C_DIS
LIN {X -12.0742,Y 11.5848,Z 56,A 129.1233,B 24.7922,C -3.3235,E1 24.8829,E2 -406.7925} C_DIS
LIN {X -12.994,Y 10.5426,Z 56,A 134.4151,B 24.7935,C -3.3133,E1 24.8734,E2 -412.0839} C_DIS
LIN {X -13.9005,Y 9.3152,Z 56,A 139.6246,B 24.7952,C -3.2994,E1 24.865,E2 -417.2856} C_DIS
LIN {X -14.6588,Y 8.0688,Z 56,A 144.2201,B 24.7971,C -3.2844,E1 24.8586,E2 -421.8691} C_DIS
LIN {X -15.2198,Y 6.954,Z 56,A 149.1516,B 24.7984,C -3.2738,E1 24.8526,E2 -426.8019} C_DIS
LIN {X -15.7547,Y 5.6375,Z 56,A 153.975,B 24.8002,C -3.2592,E1 24.8479,E2 -431.6175} C_DIS
LIN {X -16.209,Y 4.1546,Z 56,A 159.4531,B 24.8021,C -3.2435,E1 24.8438,E2 -437.0897} C_DIS
LIN {X -16.5365,Y 2.5566,Z 56,A 164.297,B 24.8045,C -3.2244,E1 24.8414,E2 -441.9166} C_DIS
LIN {X -16.6738,Y 1.4046,Z 56,A 168.9454,B 24.8058,C -3.2137,E1 24.8401,E2 -446.5672} C_DIS
LIN {X -16.7316,Y 0.1235,Z 56,A 172.775,B 24.8076,C -3.1987,E1 24.8398,E2 -450.3839} C_DIS
LIN {X -16.6916,Y -1.1558,Z 56,A 177.1549,B 24.8092,C -3.1852,E1 24.8403,E2 -454.7577} C_DIS
LIN {X -16.5559,Y -2.4288,Z 56,A -178.1385,B 24.8107,C -3.1725,E1 24.8419,E2 -459.4622} C_DIS
LIN {X -16.3409,Y -3.6012,Z 56,A -173.9484,B 24.8122,C -3.1606,E1 24.8443,E2 -463.6483} C_DIS
LIN {X -16.0261,Y -4.8127,Z 56,A -169.3021,B 24.8135,C -3.149,E1 24.8478,E2 -468.2937} C_DIS
LIN {X -15.4804,Y -6.3506,Z 56,A -164.196,B 24.8156,C -3.1319,E1 24.8528,E2 -473.3876} C_DIS
LIN {X -14.9878,Y -7.4401,Z 56,A -160.1903,B 24.8169,C -3.1205,E1 24.8576,E2 -477.3878} C_DIS
LIN {X -14.543,Y -8.2759,Z 56,A -156.1365,B 24.8176,C -3.1144,E1 24.8631,E2 -481.4483} C_DIS
LIN {X -13.4232,Y -9.9907,Z 56,A -149.333,B 24.8197,C -3.0967,E1 24.8739,E2 -488.243} C_DIS
LIN {X -12.4747,Y -11.1522,Z 56,A -144.7685,B 24.8213,C -3.0834,E1 24.8822,E2 -492.7965} C_DIS
LIN {X -11.6467,Y -12.0146,Z 56,A -140.1888,B 24.822,C -3.0767,E1 24.8912,E2 -497.3796} C_DIS
LIN {X -10.4142,Y -13.0973,Z 56,A -134.2429,B 24.8231,C -3.0677,E1 24.9039,E2 -503.3269} C_DIS
LIN {X -8.8311,Y -14.2122,Z 56,A -126.7298,B 24.8238,C -3.0613,E1 24.9215,E2 -510.8492} C_DIS
LIN {X -6.9587,Y -15.2176,Z 56,A -119.8099,B 24.825,C -3.0512,E1 24.9388,E2 -517.7629} C_DIS
LIN {X -5.1204,Y -15.9302,Z 56,A -113.6946,B 24.826,C -3.0426,E1 24.9549,E2 -523.8696} C_DIS
LIN {X -3.3841,Y -16.3872,Z 56,A -108.2439,B 24.8268,C -3.0358,E1 24.9696,E2 -529.3119} C_DIS
LIN {X -2.2946,Y -16.575,Z 56,A -103.4609,B 24.8263,C -3.0403,E1 24.9829,E2 -534.1095} C_DIS
LIN {X -0.4674,Y -16.7265,Z 56,A -97.3163,B 24.8263,C -3.0398,E1 25,E2 -540.2549} C_DIS
LIN {X -0.4674,Y -16.7265,Z 56,A -97.3163,B 24.8263,C -3.0398,E1 25,E2 -540.2549} C_DIS
Enddeposition()
LIN {X 0.078,Y -15.7325,Z 56,A -98.1107,B 24.826,C -3.0426,E1 24.9978,E2 -539.4672} C_DIS
Startdeposition()
$VEL.CP = VEL_PRINT
LIN {X -1.0725,Y -15.6983,Z 56,A -102.5995,B 24.8262,C -3.0408,E1 24.9853,E2 -534.9727} C_DIS
LIN {X -2.7791,Y -15.4876,Z 56,A -108.5568,B 24.8259,C -3.0437,E1 24.9688,E2 -529.0174} C_DIS
LIN {X -3.8605,Y -15.2542,Z 56,A -112.4491,B 24.8256,C -3.0463,E1 24.9583,E2 -525.1262} C_DIS
LIN {X -4.8776,Y -14.96,Z 56,A -116.8935,B 24.8256,C -3.0465,E1 24.9464,E2 -520.6744} C_DIS
LIN {X -6.5904,Y -14.2885,Z 56,A -122.7481,B 24.8244,C -3.0566,E1 24.9313,E2 -514.8304} C_DIS
LIN {X -7.7686,Y -13.6834,Z 56,A -128.3627,B 24.824,C -3.0597,E1 24.9175,E2 -509.2077} C_DIS
LIN {X -8.9617,Y -12.9334,Z 56,A -133.2009,B 24.823,C -3.0686,E1 24.9063,E2 -504.3747} C_DIS
LIN {X -9.826,Y -12.2896,Z 56,A -138.5969,B 24.8227,C -3.0708,E1 24.8945,E2 -498.9639} C_DIS
LIN {X -11.9516,Y -10.2347,Z 56,A -147.7873,B 24.8196,C -3.0978,E1 24.8767,E2 -489.7985} C_DIS
LIN {X -12.9034,Y -9.0047,Z 56,A -153.9187,B 24.8182,C -3.1099,E1 24.8665,E2 -483.6666} C_DIS
LIN {X -13.6281,Y -7.8651,Z 56,A -158.6371,B 24.8166,C -3.1229,E1 24.8597,E2 -478.9552} C_DIS
LIN {X -14.0791,Y -7.0263,Z 56,A -163.3921,B 24.8159,C -3.1293,E1 24.8537,E2 -474.1898} C_DIS
LIN {X -15.0367,Y -4.6356,Z 56,A -171.4295,B 24.8124,C -3.1588,E1 24.8461,E2 -466.1777} C_DIS
LIN {X -15.3616,Y -3.4082,Z 56,A -175.6167,B 24.8106,C -3.1734,E1 24.8433,E2 -462.001} C_DIS
LIN {X -15.6099,Y -1.9759,Z 56,A 178.1225,B 24.8089,C -3.1876,E1 24.8406,E2 -455.7369} C_DIS
LIN {X -15.732,Y -0.279,Z 56,A 171.3982,B 24.8067,C -3.2058,E1 24.8398,E2 -449.0157} C_DIS
LIN {X -15.6473,Y 1.6581,Z 56,A 165.4964,B 24.8038,C -3.2299,E1 24.8409,E2 -443.1362} C_DIS
LIN {X -15.536,Y 2.4962,Z 56,A 161.8652,B 24.8028,C -3.2384,E1 24.8424,E2 -439.5038} C_DIS
LIN {X -15.2315,Y 3.949,Z 56,A 156.833,B 24.8006,C -3.2557,E1 24.8456,E2 -434.4835} C_DIS
LIN {X -14.9697,Y 4.8476,Z 56,A 152.8368,B 24.7995,C -3.2648,E1 24.8489,E2 -430.4862} C_DIS
LIN {X -14.3879,Y 6.3707,Z 56,A 147.609,B 24.7972,C -3.2838,E1 24.8544,E2 -425.2748} C_DIS
LIN {X -13.8058,Y 7.5495,Z 56,A 141.5309,B 24.7958,C -3.2946,E1 24.8622,E2 -419.1903} C_DIS
LIN {X -12.6087,Y 9.4135,Z 56,A 133.6317,B 24.7931,C -3.3165,E1 24.8747,E2 -411.3045} C_DIS
LIN {X -11.873,Y 10.3257,Z 56,A 129.7388,B 24.7916,C -3.3281,E1 24.8817,E2 -407.4215} C_DIS
LIN {X -10.5919,Y 11.6363,Z 56,A 122.7366,B 24.7898,C -3.3426,E1 24.8957,E2 -400.4248} C_DIS
LIN {X -9.7542,Y 12.3469,Z 56,A 118.9884,B 24.7886,C -3.3517,E1 24.9039,E2 -396.6844} C_DIS
LIN {X -8.7655,Y 13.0674,Z 56,A 114.6243,B 24.7875,C -3.3605,E1 24.9139,E2 -392.3266} C_DIS
LIN {X -7.9189,Y 13.5974,Z 56,A 110.1425,B 24.787,C -3.3641,E1 24.9247,E2 -387.84} C_DIS
LIN {X -6.0431,Y 14.5281,Z 56,A 104.1257,B 24.7849,C -3.3811,E1 24.9398,E2 -381.8487} C_DIS
LIN {X -5.1695,Y 14.8615,Z 56,A 99.8423,B 24.7848,C -3.382,E1 24.9511,E2 -377.5588} C_DIS
LIN {X -3.8473,Y 15.2576,Z 56,A 94.8849,B 24.7841,C -3.3874,E1 24.9644,E2 -372.6065} C_DIS
LIN {X -2.4706,Y 15.5399,Z 56,A 89.635,B 24.7837,C -3.3906,E1 24.9788,E2 -367.3589} C_DIS
LIN {X -1.1398,Y 15.6936,Z 56,A 84.8955,B 24.7833,C -3.3936,E1 24.992,E2 -362.624} C_DIS
LIN {X -0.0813,Y 15.7348,Z 56,A 80.8405,B 24.7833,C -3.3936,E1 25.0033,E2 -358.5688} C_DIS
LIN {X 1.4955,Y 15.6635,Z 56,A 75.5691,B 24.783,C -3.3959,E1 25.018,E2 -353.3052} C_DIS
LIN {X 2.7899,Y 15.4857,Z 56,A 70.2184,B 24.7836,C -3.3914,E1 25.0327,E2 -347.9489} C_DIS
LIN {X 3.819,Y 15.2648,Z 56,A 66.0833,B 24.7841,C -3.3876,E1 25.0439,E2 -343.8108} C_DIS
LIN {X 5.266,Y 14.8277,Z 56,A 60.8193,B 24.7844,C -3.3846,E1 25.0579,E2 -338.5498} C_DIS
LIN {X 6.6402,Y 14.2653,Z 56,A 56.1966,B 24.7846,C -3.3836,E1 25.0697,E2 -333.9359} C_DIS
LIN {X 7.3959,Y 13.8887,Z 56,A 52.9962,B 24.7852,C -3.379,E1 25.0776,E2 -330.7334} C_DIS
LIN {X 8.4493,Y 13.2742,Z 56,A 48.3122,B 24.7862,C -3.371,E1 25.0888,E2 -326.045} C_DIS
LIN {X 9.6725,Y 12.4111,Z 56,A 42.5649,B 24.7876,C -3.3598,E1 25.1017,E2 -320.2917} C_DIS
LIN {X 10.9009,Y 11.3473,Z 56,A 36.7429,B 24.789,C -3.3489,E1 25.1137,E2 -314.4674} C_DIS
LIN {X 11.7407,Y 10.4758,Z 56,A 31.6352,B 24.7908,C -3.3344,E1 25.1233,E2 -309.3478} C_DIS
LIN {X 13.1442,Y 8.6498,Z 56,A 23.8185,B 24.7928,C -3.3184,E1 25.136,E2 -301.5311} C_DIS
LIN {X 14.1086,Y 6.966,Z 56,A 17.3497,B 24.7946,C -3.3044,E1 25.1446,E2 -295.063} C_DIS
LIN {X 14.6386,Y 5.7708,Z 56,A 11.746,B 24.7971,C -3.2845,E1 25.1506,E2 -289.4429} C_DIS
LIN {X 15.2091,Y 4.0335,Z 56,A 5.8718,B 24.7987,C -3.2713,E1 25.1553,E2 -283.571} C_DIS
LIN {X 15.5107,Y 2.6454,Z 56,A 0.7035,B 24.8006,C -3.2558,E1 25.158,E2 -278.3961} C_DIS
LIN {X 15.6835,Y 1.2697,Z 56,A -4.4781,B 24.8027,C -3.2392,E1 25.1595,E2 -273.2058} C_DIS
LIN {X 15.7342,Y -0.199,Z 56,A -10.0506,B 24.8049,C -3.2208,E1 25.1596,E2 -267.6228} C_DIS
LIN {X 15.584,Y -2.1754,Z 56,A -16.2067,B 24.8066,C -3.207,E1 25.158,E2 -261.4705} C_DIS
LIN {X 15.2408,Y -3.9126,Z 56,A -24.2634,B 24.8105,C -3.1741,E1 25.1531,E2 -253.3826} C_DIS
Enddeposition()
END
